   "LIST_CODE_CHAR".Contain_In_Bath11 := "LIST_CODE_CHAR".Contain_In_Bath10;
   "LIST_CODE_CHAR".Contain_In_Bath10 := "LIST_CODE_CHAR".Contain_In_Bath9;
   "LIST_CODE_CHAR".Contain_In_Bath9 := "LIST_CODE_CHAR".Contain_In_Bath8;
   "LIST_CODE_CHAR".Contain_In_Bath8 := "LIST_CODE_CHAR".Contain_In_Bath7;
   "LIST_CODE_CHAR".Contain_In_Bath7 := "LIST_CODE_CHAR".Contain_In_Bath6;
   IF "LIST_CODE_CHAR".Contain_In_Bath6.Barcode_P1 <> '' OR "LIST_CODE_CHAR".Contain_In_Bath6.Barcode_P2 <> '' THEN
       ;
       "LIST_CODE_CHAR".Contain_In_Bath6.Barcode_P1 := '';
       "LIST_CODE_CHAR".Contain_In_Bath6.Barcode_P2 := '';
   END_IF;
   IF "LIST_CODE_CHAR".Contain_In_Bath11.Barcode_P1 <> '' THEN
       ;
       "TCP_PARAMETER".DATA := 'd';
       "SEND_TCP_TRIGGER_1" := TRUE;
   END_IF;


   //Area Robot
   IF "LIST_CODE_CHAR".Contain_In_Bath3.Barcode_P2 = '1' THEN
       ;
       "LIST_CODE_CHAR".Barcode_Queue_Robot := "LIST_CODE_CHAR".Contain_In_Bath3;// Pick to bath 6
       "RUN_TIME_PARAM".REQUEST_PICK_TYPE := 1;
   ELSIF "LIST_CODE_CHAR".Contain_In_Bath3.Barcode_P2 = '2' OR "LIST_CODE_CHAR".Contain_In_Bath3.Barcode_P2 = '3' THEN
       ;
       "LIST_CODE_CHAR".Barcode_Queue_Robot := "LIST_CODE_CHAR".Contain_In_Bath3;// At Bath 4
       "RUN_TIME_PARAM".REQUEST_PICK_TYPE := 3;
   ELSIF "LIST_CODE_CHAR".Contain_In_Bath3.Barcode_P2 = '4' THEN
       ;
       "LIST_CODE_CHAR".Barcode_Queue_Robot := "LIST_CODE_CHAR".Contain_In_Bath3;// Pick To Bath 5
       "RUN_TIME_PARAM".REQUEST_PICK_TYPE := 2;
   ELSE
       "LIST_CODE_CHAR".Barcode_Queue_Robot.Barcode_P1 := '';
       "LIST_CODE_CHAR".Barcode_Queue_Robot.Barcode_P2 := '';
       "RUN_TIME_PARAM".REQUEST_PICK_TYPE := 0;
       ;
   END_IF;

   "LIST_CODE_CHAR".Contain_In_Bath3 := "LIST_CODE_CHAR".Contain_In_Bath2;
   "LIST_CODE_CHAR".Contain_In_Bath2 := "LIST_CODE_CHAR".Contain_In_Bath1;

   // Area 1
   IF "DETECT_VALUE".SCANED_BARCODE <> '' AND "SS Up XL Nâng Input" = TRUE THEN
       ;
       "QUEUE_TO_RUN_BARCODE"(Scaned_Barcode:="DETECT_VALUE".SCANED_BARCODE,OUT_OF_BARCODE=> #Check_Has_Barcode);

   ELSE
       ;
       "LIST_CODE_CHAR".Contain_In_Bath1.Barcode_P1 := '';
       "LIST_CODE_CHAR".Contain_In_Bath1.Barcode_P2 := '';
   END_IF;

   IF #Check_Has_Barcode = TRUE THEN
       ;
       "TCP_PARAMETER".DATA := 'e'; // Khi Không còn barcode trong hàng chờ
       "SEND_TCP_TRIGGER" := TRUE;
   END_IF;
END_FUNCTION

FUNCTION "CONTROL_WATER_PUMP" : Void   // FC2, LAD
{ S7_Optimized_Access := 'TRUE' }
VERSION : 0.1
   VAR_TEMP   // added for the SCL form of the ladder/FBD networks
      _w1 : Bool;
   END_VAR
BEGIN

REGION Network 1: TANK 1
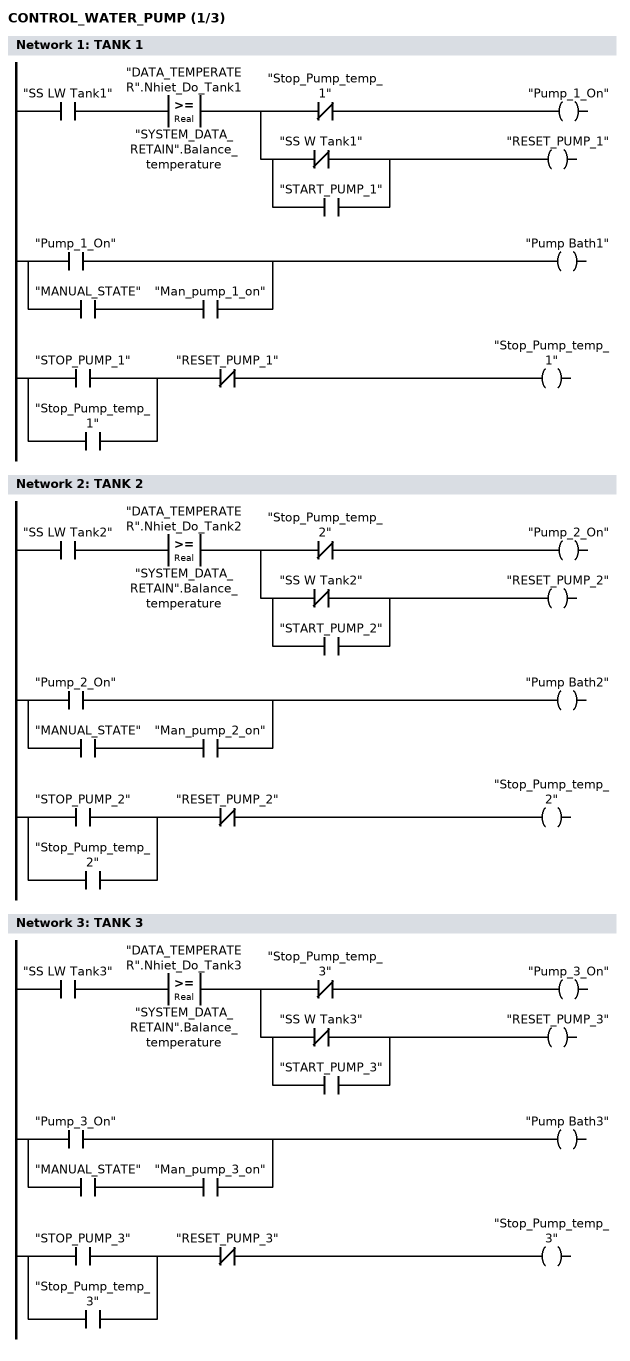
   RUNG wire#powerrail
      Contact( "SS LW Tank1" )
      { S7_Templates := "SrcType := Real" } GE_Contact(in1 := "DATA_TEMPERATER".Nhiet_Do_Tank1, in2 := "SYSTEM_DATA_RETAIN".Balance_temperature)
      wire#w1
      I_Contact( "Stop_Pump_temp_1" )
      Coil( "Pump_1_On" )
   END_RUNG
   RUNG wire#w1
      I_Contact( "SS W Tank1" )
      wire#w2
      Coil( "RESET_PUMP_1" )
   END_RUNG
   RUNG wire#w1
      Contact( "START_PUMP_1" )
   END_RUNG wire#w2
   RUNG wire#powerrail
      Contact( "Pump_1_On" )
      wire#w3
      Coil( "Pump Bath1" )
   END_RUNG
   RUNG wire#powerrail
      Contact( "MANUAL_STATE" )
      Contact( "Man_pump_1_on" )
   END_RUNG wire#w3
   RUNG wire#powerrail
      Contact( "STOP_PUMP_1" )
      wire#w4
      I_Contact( "RESET_PUMP_1" )
      Coil( "Stop_Pump_temp_1" )
   END_RUNG
   RUNG wire#powerrail
      Contact( "Stop_Pump_temp_1" )
   END_RUNG wire#w4
   // the same network as SCL:
   #_w1 := "SS LW Tank1" AND ("DATA_TEMPERATER".Nhiet_Do_Tank1 >= "SYSTEM_DATA_RETAIN".Balance_temperature);
   "Pump_1_On" := #_w1 AND NOT "Stop_Pump_temp_1";
   "RESET_PUMP_1" := #_w1 AND (NOT "SS W Tank1" OR "START_PUMP_1");
   "Pump Bath1" := "Pump_1_On" OR ("MANUAL_STATE" AND "Man_pump_1_on");
   "Stop_Pump_temp_1" := ("STOP_PUMP_1" OR "Stop_Pump_temp_1") AND NOT "RESET_PUMP_1";
END_REGION

REGION Network 2: TANK 2
   RUNG wire#powerrail
      Contact( "SS LW Tank2" )
      { S7_Templates := "SrcType := Real" } GE_Contact(in1 := "DATA_TEMPERATER".Nhiet_Do_Tank2, in2 := "SYSTEM_DATA_RETAIN".Balance_temperature)
      wire#w1
      I_Contact( "Stop_Pump_temp_2" )
      Coil( "Pump_2_On" )
   END_RUNG
   RUNG wire#w1
      I_Contact( "SS W Tank2" )
      wire#w2
      Coil( "RESET_PUMP_2" )
   END_RUNG
   RUNG wire#w1
      Contact( "START_PUMP_2" )
   END_RUNG wire#w2
   RUNG wire#powerrail
      Contact( "Pump_2_On" )
      wire#w3
      Coil( "Pump Bath2" )
   END_RUNG
   RUNG wire#powerrail
      Contact( "MANUAL_STATE" )
      Contact( "Man_pump_2_on" )
   END_RUNG wire#w3
   RUNG wire#powerrail
      Contact( "STOP_PUMP_2" )
      wire#w4
      I_Contact( "RESET_PUMP_2" )
      Coil( "Stop_Pump_temp_2" )
   END_RUNG
   RUNG wire#powerrail
      Contact( "Stop_Pump_temp_2" )
   END_RUNG wire#w4
   // the same network as SCL:
   #_w1 := "SS LW Tank2" AND ("DATA_TEMPERATER".Nhiet_Do_Tank2 >= "SYSTEM_DATA_RETAIN".Balance_temperature);
   "Pump_2_On" := #_w1 AND NOT "Stop_Pump_temp_2";
   "RESET_PUMP_2" := #_w1 AND (NOT "SS W Tank2" OR "START_PUMP_2");
   "Pump Bath2" := "Pump_2_On" OR ("MANUAL_STATE" AND "Man_pump_2_on");
   "Stop_Pump_temp_2" := ("STOP_PUMP_2" OR "Stop_Pump_temp_2") AND NOT "RESET_PUMP_2";
END_REGION

REGION Network 3: TANK 3
   RUNG wire#powerrail
      Contact( "SS LW Tank3" )
      { S7_Templates := "SrcType := Real" } GE_Contact(in1 := "DATA_TEMPERATER".Nhiet_Do_Tank3, in2 := "SYSTEM_DATA_RETAIN".Balance_temperature)
      wire#w1
      I_Contact( "Stop_Pump_temp_3" )
      Coil( "Pump_3_On" )
   END_RUNG
   RUNG wire#w1
      I_Contact( "SS W Tank3" )
      wire#w2
      Coil( "RESET_PUMP_3" )
   END_RUNG
   RUNG wire#w1
      Contact( "START_PUMP_3" )
   END_RUNG wire#w2
   RUNG wire#powerrail
      Contact( "Pump_3_On" )
      wire#w3
      Coil( "Pump Bath3" )
   END_RUNG
   RUNG wire#powerrail
      Contact( "MANUAL_STATE" )
      Contact( "Man_pump_3_on" )
   END_RUNG wire#w3
   RUNG wire#powerrail
      Contact( "STOP_PUMP_3" )
      wire#w4
      I_Contact( "RESET_PUMP_3" )
      Coil( "Stop_Pump_temp_3" )
   END_RUNG
   RUNG wire#powerrail
      Contact( "Stop_Pump_temp_3" )
   END_RUNG wire#w4
   // the same network as SCL:
   #_w1 := "SS LW Tank3" AND ("DATA_TEMPERATER".Nhiet_Do_Tank3 >= "SYSTEM_DATA_RETAIN".Balance_temperature);
   "Pump_3_On" := #_w1 AND NOT "Stop_Pump_temp_3";
   "RESET_PUMP_3" := #_w1 AND (NOT "SS W Tank3" OR "START_PUMP_3");
   "Pump Bath3" := "Pump_3_On" OR ("MANUAL_STATE" AND "Man_pump_3_on");
   "Stop_Pump_temp_3" := ("STOP_PUMP_3" OR "Stop_Pump_temp_3") AND NOT "RESET_PUMP_3";
END_REGION

REGION Network 4: TANK 4
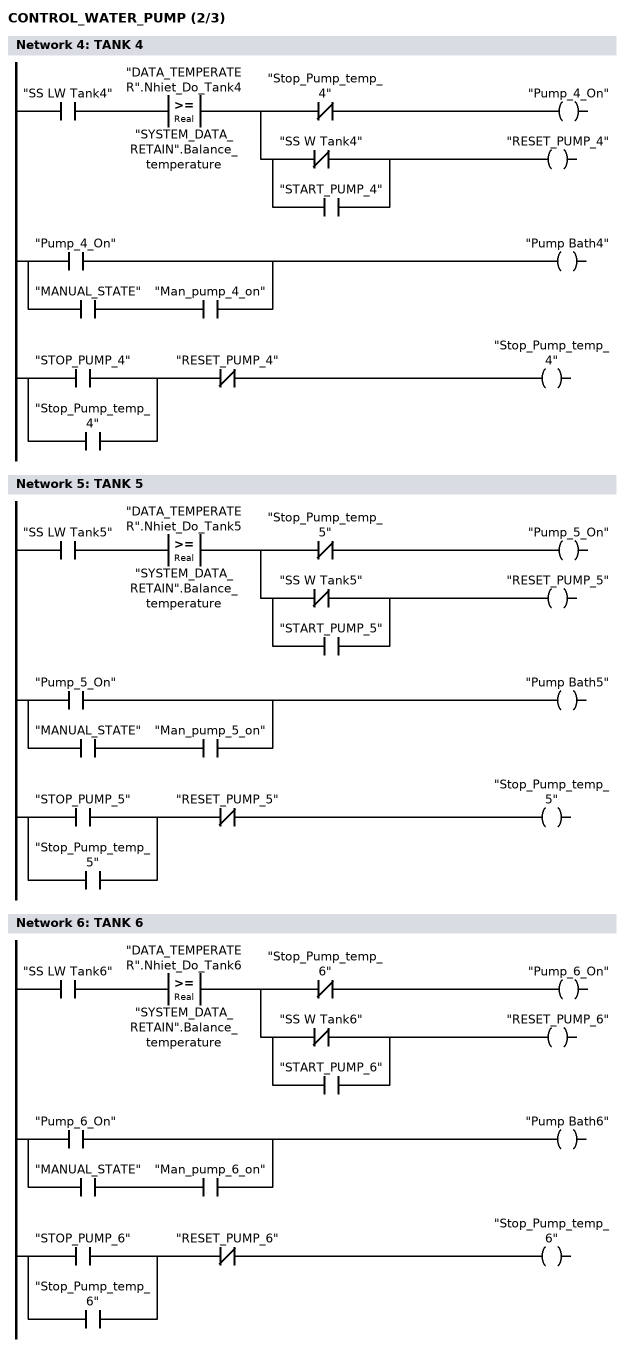
   RUNG wire#powerrail
      Contact( "SS LW Tank4" )
      { S7_Templates := "SrcType := Real" } GE_Contact(in1 := "DATA_TEMPERATER".Nhiet_Do_Tank4, in2 := "SYSTEM_DATA_RETAIN".Balance_temperature)
      wire#w1
      I_Contact( "Stop_Pump_temp_4" )
      Coil( "Pump_4_On" )
   END_RUNG
   RUNG wire#w1
      I_Contact( "SS W Tank4" )
      wire#w2
      Coil( "RESET_PUMP_4" )
   END_RUNG
   RUNG wire#w1
      Contact( "START_PUMP_4" )
   END_RUNG wire#w2
   RUNG wire#powerrail
      Contact( "Pump_4_On" )
      wire#w3
      Coil( "Pump Bath4" )
   END_RUNG
   RUNG wire#powerrail
      Contact( "MANUAL_STATE" )
      Contact( "Man_pump_4_on" )
   END_RUNG wire#w3
   RUNG wire#powerrail
      Contact( "STOP_PUMP_4" )
      wire#w4
      I_Contact( "RESET_PUMP_4" )
      Coil( "Stop_Pump_temp_4" )
   END_RUNG
   RUNG wire#powerrail
      Contact( "Stop_Pump_temp_4" )
   END_RUNG wire#w4
   // the same network as SCL:
   #_w1 := "SS LW Tank4" AND ("DATA_TEMPERATER".Nhiet_Do_Tank4 >= "SYSTEM_DATA_RETAIN".Balance_temperature);
   "Pump_4_On" := #_w1 AND NOT "Stop_Pump_temp_4";
   "RESET_PUMP_4" := #_w1 AND (NOT "SS W Tank4" OR "START_PUMP_4");
   "Pump Bath4" := "Pump_4_On" OR ("MANUAL_STATE" AND "Man_pump_4_on");
   "Stop_Pump_temp_4" := ("STOP_PUMP_4" OR "Stop_Pump_temp_4") AND NOT "RESET_PUMP_4";
END_REGION

REGION Network 5: TANK 5
   RUNG wire#powerrail
      Contact( "SS LW Tank5" )
      { S7_Templates := "SrcType := Real" } GE_Contact(in1 := "DATA_TEMPERATER".Nhiet_Do_Tank5, in2 := "SYSTEM_DATA_RETAIN".Balance_temperature)
      wire#w1
      I_Contact( "Stop_Pump_temp_5" )
      Coil( "Pump_5_On" )
   END_RUNG
   RUNG wire#w1
      I_Contact( "SS W Tank5" )
      wire#w2
      Coil( "RESET_PUMP_5" )
   END_RUNG
   RUNG wire#w1
      Contact( "START_PUMP_5" )
   END_RUNG wire#w2
   RUNG wire#powerrail
      Contact( "Pump_5_On" )
      wire#w3
      Coil( "Pump Bath5" )
   END_RUNG
   RUNG wire#powerrail
      Contact( "MANUAL_STATE" )
      Contact( "Man_pump_5_on" )
   END_RUNG wire#w3
   RUNG wire#powerrail
      Contact( "STOP_PUMP_5" )
      wire#w4
      I_Contact( "RESET_PUMP_5" )
      Coil( "Stop_Pump_temp_5" )
   END_RUNG
   RUNG wire#powerrail
      Contact( "Stop_Pump_temp_5" )
   END_RUNG wire#w4
   // the same network as SCL:
   #_w1 := "SS LW Tank5" AND ("DATA_TEMPERATER".Nhiet_Do_Tank5 >= "SYSTEM_DATA_RETAIN".Balance_temperature);
   "Pump_5_On" := #_w1 AND NOT "Stop_Pump_temp_5";
   "RESET_PUMP_5" := #_w1 AND (NOT "SS W Tank5" OR "START_PUMP_5");
   "Pump Bath5" := "Pump_5_On" OR ("MANUAL_STATE" AND "Man_pump_5_on");
   "Stop_Pump_temp_5" := ("STOP_PUMP_5" OR "Stop_Pump_temp_5") AND NOT "RESET_PUMP_5";
END_REGION

REGION Network 6: TANK 6
   RUNG wire#powerrail
      Contact( "SS LW Tank6" )
      { S7_Templates := "SrcType := Real" } GE_Contact(in1 := "DATA_TEMPERATER".Nhiet_Do_Tank6, in2 := "SYSTEM_DATA_RETAIN".Balance_temperature)
      wire#w1
      I_Contact( "Stop_Pump_temp_6" )
      Coil( "Pump_6_On" )
   END_RUNG
   RUNG wire#w1
      I_Contact( "SS W Tank6" )
      wire#w2
      Coil( "RESET_PUMP_6" )
   END_RUNG
   RUNG wire#w1
      Contact( "START_PUMP_6" )
   END_RUNG wire#w2
   RUNG wire#powerrail
      Contact( "Pump_6_On" )
      wire#w3
      Coil( "Pump Bath6" )
   END_RUNG
   RUNG wire#powerrail
      Contact( "MANUAL_STATE" )
      Contact( "Man_pump_6_on" )
   END_RUNG wire#w3
   RUNG wire#powerrail
      Contact( "STOP_PUMP_6" )
      wire#w4
      I_Contact( "RESET_PUMP_6" )
      Coil( "Stop_Pump_temp_6" )
   END_RUNG
   RUNG wire#powerrail
      Contact( "Stop_Pump_temp_6" )
   END_RUNG wire#w4
   // the same network as SCL:
   #_w1 := "SS LW Tank6" AND ("DATA_TEMPERATER".Nhiet_Do_Tank6 >= "SYSTEM_DATA_RETAIN".Balance_temperature);
   "Pump_6_On" := #_w1 AND NOT "Stop_Pump_temp_6";
   "RESET_PUMP_6" := #_w1 AND (NOT "SS W Tank6" OR "START_PUMP_6");
   "Pump Bath6" := "Pump_6_On" OR ("MANUAL_STATE" AND "Man_pump_6_on");
   "Stop_Pump_temp_6" := ("STOP_PUMP_6" OR "Stop_Pump_temp_6") AND NOT "RESET_PUMP_6";
END_REGION

REGION Network 7: TANK 7
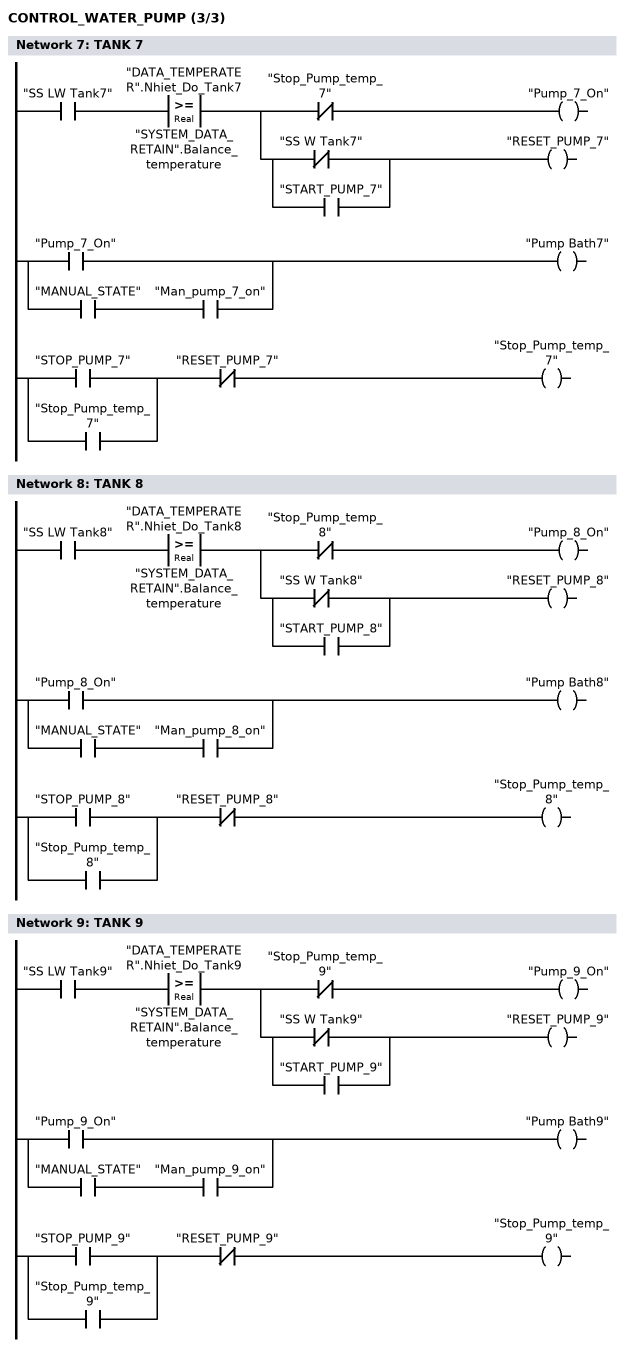
   RUNG wire#powerrail
      Contact( "SS LW Tank7" )
      { S7_Templates := "SrcType := Real" } GE_Contact(in1 := "DATA_TEMPERATER".Nhiet_Do_Tank7, in2 := "SYSTEM_DATA_RETAIN".Balance_temperature)
      wire#w1
      I_Contact( "Stop_Pump_temp_7" )
      Coil( "Pump_7_On" )
   END_RUNG
   RUNG wire#w1
      I_Contact( "SS W Tank7" )
      wire#w2
      Coil( "RESET_PUMP_7" )
   END_RUNG
   RUNG wire#w1
      Contact( "START_PUMP_7" )
   END_RUNG wire#w2
   RUNG wire#powerrail
      Contact( "Pump_7_On" )
      wire#w3
      Coil( "Pump Bath7" )
   END_RUNG
   RUNG wire#powerrail
      Contact( "MANUAL_STATE" )
      Contact( "Man_pump_7_on" )
   END_RUNG wire#w3
   RUNG wire#powerrail
      Contact( "STOP_PUMP_7" )
      wire#w4
      I_Contact( "RESET_PUMP_7" )
      Coil( "Stop_Pump_temp_7" )
   END_RUNG
   RUNG wire#powerrail
      Contact( "Stop_Pump_temp_7" )
   END_RUNG wire#w4
   // the same network as SCL:
   #_w1 := "SS LW Tank7" AND ("DATA_TEMPERATER".Nhiet_Do_Tank7 >= "SYSTEM_DATA_RETAIN".Balance_temperature);
   "Pump_7_On" := #_w1 AND NOT "Stop_Pump_temp_7";
   "RESET_PUMP_7" := #_w1 AND (NOT "SS W Tank7" OR "START_PUMP_7");
   "Pump Bath7" := "Pump_7_On" OR ("MANUAL_STATE" AND "Man_pump_7_on");
   "Stop_Pump_temp_7" := ("STOP_PUMP_7" OR "Stop_Pump_temp_7") AND NOT "RESET_PUMP_7";
END_REGION

REGION Network 8: TANK 8
   RUNG wire#powerrail
      Contact( "SS LW Tank8" )
      { S7_Templates := "SrcType := Real" } GE_Contact(in1 := "DATA_TEMPERATER".Nhiet_Do_Tank8, in2 := "SYSTEM_DATA_RETAIN".Balance_temperature)
      wire#w1
      I_Contact( "Stop_Pump_temp_8" )
      Coil( "Pump_8_On" )
   END_RUNG
   RUNG wire#w1
      I_Contact( "SS W Tank8" )
      wire#w2
      Coil( "RESET_PUMP_8" )
   END_RUNG
   RUNG wire#w1
      Contact( "START_PUMP_8" )
   END_RUNG wire#w2
   RUNG wire#powerrail
      Contact( "Pump_8_On" )
      wire#w3
      Coil( "Pump Bath8" )
   END_RUNG
   RUNG wire#powerrail
      Contact( "MANUAL_STATE" )
      Contact( "Man_pump_8_on" )
   END_RUNG wire#w3
   RUNG wire#powerrail
      Contact( "STOP_PUMP_8" )
      wire#w4
      I_Contact( "RESET_PUMP_8" )
      Coil( "Stop_Pump_temp_8" )
   END_RUNG
   RUNG wire#powerrail
      Contact( "Stop_Pump_temp_8" )
   END_RUNG wire#w4
   // the same network as SCL:
   #_w1 := "SS LW Tank8" AND ("DATA_TEMPERATER".Nhiet_Do_Tank8 >= "SYSTEM_DATA_RETAIN".Balance_temperature);
   "Pump_8_On" := #_w1 AND NOT "Stop_Pump_temp_8";
   "RESET_PUMP_8" := #_w1 AND (NOT "SS W Tank8" OR "START_PUMP_8");
   "Pump Bath8" := "Pump_8_On" OR ("MANUAL_STATE" AND "Man_pump_8_on");
   "Stop_Pump_temp_8" := ("STOP_PUMP_8" OR "Stop_Pump_temp_8") AND NOT "RESET_PUMP_8";
END_REGION

REGION Network 9: TANK 9
   RUNG wire#powerrail
      Contact( "SS LW Tank9" )
      { S7_Templates := "SrcType := Real" } GE_Contact(in1 := "DATA_TEMPERATER".Nhiet_Do_Tank9, in2 := "SYSTEM_DATA_RETAIN".Balance_temperature)
      wire#w1
      I_Contact( "Stop_Pump_temp_9" )
      Coil( "Pump_9_On" )
   END_RUNG
   RUNG wire#w1
      I_Contact( "SS W Tank9" )
      wire#w2
      Coil( "RESET_PUMP_9" )
   END_RUNG
   RUNG wire#w1
      Contact( "START_PUMP_9" )
   END_RUNG wire#w2
   RUNG wire#powerrail
      Contact( "Pump_9_On" )
      wire#w3
      Coil( "Pump Bath9" )
   END_RUNG
   RUNG wire#powerrail
      Contact( "MANUAL_STATE" )
      Contact( "Man_pump_9_on" )
   END_RUNG wire#w3
   RUNG wire#powerrail
      Contact( "STOP_PUMP_9" )
      wire#w4
      I_Contact( "RESET_PUMP_9" )
      Coil( "Stop_Pump_temp_9" )
   END_RUNG
   RUNG wire#powerrail
      Contact( "Stop_Pump_temp_9" )
   END_RUNG wire#w4
   // the same network as SCL:
   #_w1 := "SS LW Tank9" AND ("DATA_TEMPERATER".Nhiet_Do_Tank9 >= "SYSTEM_DATA_RETAIN".Balance_temperature);
   "Pump_9_On" := #_w1 AND NOT "Stop_Pump_temp_9";
   "RESET_PUMP_9" := #_w1 AND (NOT "SS W Tank9" OR "START_PUMP_9");
   "Pump Bath9" := "Pump_9_On" OR ("MANUAL_STATE" AND "Man_pump_9_on");
   "Stop_Pump_temp_9" := ("STOP_PUMP_9" OR "Stop_Pump_temp_9") AND NOT "RESET_PUMP_9";
END_REGION
END_FUNCTION

FUNCTION "Move_BarCode_Data" : Void   // FC3, SCL
{ S7_Optimized_Access := 'TRUE' }
VERSION : 0.1
BEGIN
END_FUNCTION

FUNCTION "INT_TO_BIT_ARRAY" : Void   // FC5, SCL
{ S7_Optimized_Access := 'TRUE' }
VERSION : 0.1
   VAR_INPUT
      IN : Int;
   END_VAR
   VAR_OUTPUT
      OUT : Array[0..15] of Bool;
   END_VAR
   VAR_TEMP
      TEMP : Int;
      TEMPW : Word;
      TEMP_B : Int;
      DEM : Int;
      INS : Int;
   END_VAR
BEGIN
   #TEMP := #IN;
   #TEMP_B := 0;
   #TEMPW := 0;
   #DEM := 0;
   IF #IN = 0 THEN
       FOR #INS := 0 TO 15 DO
           #OUT[#INS] := FALSE;
           ;
       END_FOR;
   ELSE
       WHILE #TEMP <> 0 DO
           #TEMP_B := #TEMP MOD 2;
           #TEMP := #TEMP / 2;
           IF #TEMP_B = 1 THEN
               #OUT[#DEM] := TRUE;
               ;
           ELSIF #TEMP_B = 0 THEN
               #OUT[#DEM] := FALSE;
               ;
           END_IF;
           #DEM := #DEM + 1;
       END_WHILE;
       IF #DEM < 15 THEN
           FOR #DEM := #DEM TO 15 DO
               #OUT[#DEM] := FALSE;
           END_FOR;
       END_IF;
   END_IF;
END_FUNCTION

FUNCTION "QUEUE_TO_RUN_BARCODE" : Void   // FC6, SCL
{ S7_Optimized_Access := 'TRUE' }
VERSION : 0.1
   VAR_INPUT
      Scaned_Barcode : String;
   END_VAR
   VAR_OUTPUT
      OUT_OF_BARCODE : Bool;
   END_VAR
BEGIN
   IF #Scaned_Barcode = "LIST_CODE_CHAR".Barcode_10.Barcode_P1 THEN
       // Truyền barcode vị trí cuối cừng vào ổ chứa barcode ở bể thứ nhất
       "LIST_CODE_CHAR".Contain_In_Bath1 := "LIST_CODE_CHAR".Barcode_10;
       //Reset giá trị Barcode 10 để đẩy mã tiếp theo lên

       //Resort 
       //9->10
       IF "LIST_CODE_CHAR".Barcode_9.Barcode_P1 = '' THEN
           #OUT_OF_BARCODE := TRUE;
       ELSE
           ;
           "LIST_CODE_CHAR".Barcode_10 := "LIST_CODE_CHAR".Barcode_9;
           //8->9
           "LIST_CODE_CHAR".Barcode_9 := "LIST_CODE_CHAR".Barcode_8;
           //7->8
           "LIST_CODE_CHAR".Barcode_8 := "LIST_CODE_CHAR".Barcode_7;
           //6->7
           "LIST_CODE_CHAR".Barcode_7 := "LIST_CODE_CHAR".Barcode_6;
           //5->6
           "LIST_CODE_CHAR".Barcode_6 := "LIST_CODE_CHAR".Barcode_5;
           //4->5
           "LIST_CODE_CHAR".Barcode_5 := "LIST_CODE_CHAR".Barcode_4;
           //3->4
           "LIST_CODE_CHAR".Barcode_4 := "LIST_CODE_CHAR".Barcode_3;
           //2->3
           "LIST_CODE_CHAR".Barcode_3 := "LIST_CODE_CHAR".Barcode_2;
           //1->2
           "LIST_CODE_CHAR".Barcode_2 := "LIST_CODE_CHAR".Barcode_1;
           //''->1
           "LIST_CODE_CHAR".Barcode_1.Barcode_P1 := '';
           "LIST_CODE_CHAR".Barcode_1.Barcode_P2 := '';
           #OUT_OF_BARCODE := FALSE;
       END_IF;

   ELSIF #Scaned_Barcode = "LIST_CODE_CHAR".Barcode_9.Barcode_P1 THEN
       "LIST_CODE_CHAR".Contain_In_Bath1 := "LIST_CODE_CHAR".Barcode_9;
       //Resort
       "LIST_CODE_CHAR".Barcode_9 := "LIST_CODE_CHAR".Barcode_8;
       //7->8
       "LIST_CODE_CHAR".Barcode_8 := "LIST_CODE_CHAR".Barcode_7;
       //6->7
       "LIST_CODE_CHAR".Barcode_7 := "LIST_CODE_CHAR".Barcode_6;
       //5->6
       "LIST_CODE_CHAR".Barcode_6 := "LIST_CODE_CHAR".Barcode_5;
       //4->5
       "LIST_CODE_CHAR".Barcode_5 := "LIST_CODE_CHAR".Barcode_4;
       //3->4
       "LIST_CODE_CHAR".Barcode_4 := "LIST_CODE_CHAR".Barcode_3;
       //2->3
       "LIST_CODE_CHAR".Barcode_3 := "LIST_CODE_CHAR".Barcode_2;
       //1->2
       "LIST_CODE_CHAR".Barcode_2 := "LIST_CODE_CHAR".Barcode_1;
       //''->1
       "LIST_CODE_CHAR".Barcode_1.Barcode_P1 := '';
       "LIST_CODE_CHAR".Barcode_1.Barcode_P2 := '';
       #OUT_OF_BARCODE := FALSE;
   ELSIF #Scaned_Barcode = "LIST_CODE_CHAR".Barcode_8.Barcode_P1 THEN
       "LIST_CODE_CHAR".Contain_In_Bath1 := "LIST_CODE_CHAR".Barcode_8;
       //Resort
       //7->8
       "LIST_CODE_CHAR".Barcode_8 := "LIST_CODE_CHAR".Barcode_7;
       //6->7
       "LIST_CODE_CHAR".Barcode_7 := "LIST_CODE_CHAR".Barcode_6;
       //5->6
       "LIST_CODE_CHAR".Barcode_6 := "LIST_CODE_CHAR".Barcode_5;
       //4->5
       "LIST_CODE_CHAR".Barcode_5 := "LIST_CODE_CHAR".Barcode_4;
       //3->4
       "LIST_CODE_CHAR".Barcode_4 := "LIST_CODE_CHAR".Barcode_3;
       //2->3
       "LIST_CODE_CHAR".Barcode_3 := "LIST_CODE_CHAR".Barcode_2;
       //1->2
       "LIST_CODE_CHAR".Barcode_2 := "LIST_CODE_CHAR".Barcode_1;
       //''->1
       "LIST_CODE_CHAR".Barcode_1.Barcode_P1 := '';
       "LIST_CODE_CHAR".Barcode_1.Barcode_P2 := '';
       #OUT_OF_BARCODE := FALSE;
   ELSIF #Scaned_Barcode = "LIST_CODE_CHAR".Barcode_7.Barcode_P1 THEN
       "LIST_CODE_CHAR".Contain_In_Bath1 := "LIST_CODE_CHAR".Barcode_7;
       //Resort
       //6->7
       "LIST_CODE_CHAR".Barcode_7 := "LIST_CODE_CHAR".Barcode_6;
       //5->6
       "LIST_CODE_CHAR".Barcode_6 := "LIST_CODE_CHAR".Barcode_5;
       //4->5
       "LIST_CODE_CHAR".Barcode_5 := "LIST_CODE_CHAR".Barcode_4;
       //3->4
       "LIST_CODE_CHAR".Barcode_4 := "LIST_CODE_CHAR".Barcode_3;
       //2->3
       "LIST_CODE_CHAR".Barcode_3 := "LIST_CODE_CHAR".Barcode_2;
       //1->2
       "LIST_CODE_CHAR".Barcode_2 := "LIST_CODE_CHAR".Barcode_1;
       //''->1
       "LIST_CODE_CHAR".Barcode_1.Barcode_P1 := '';
       "LIST_CODE_CHAR".Barcode_1.Barcode_P2 := '';
       #OUT_OF_BARCODE := FALSE;
   ELSIF #Scaned_Barcode = "LIST_CODE_CHAR".Barcode_6.Barcode_P1 THEN
       "LIST_CODE_CHAR".Contain_In_Bath1 := "LIST_CODE_CHAR".Barcode_6;
       //Resort
       //5->6
       "LIST_CODE_CHAR".Barcode_6 := "LIST_CODE_CHAR".Barcode_5;
       //4->5
       "LIST_CODE_CHAR".Barcode_5 := "LIST_CODE_CHAR".Barcode_4;
       //3->4
       "LIST_CODE_CHAR".Barcode_4 := "LIST_CODE_CHAR".Barcode_3;
       //2->3
       "LIST_CODE_CHAR".Barcode_3 := "LIST_CODE_CHAR".Barcode_2;
       //1->2
       "LIST_CODE_CHAR".Barcode_2 := "LIST_CODE_CHAR".Barcode_1;
       //''->1
       "LIST_CODE_CHAR".Barcode_1.Barcode_P1 := '';
       "LIST_CODE_CHAR".Barcode_1.Barcode_P2 := '';
       #OUT_OF_BARCODE := FALSE;
   ELSIF #Scaned_Barcode = "LIST_CODE_CHAR".Barcode_5.Barcode_P1 THEN
       "LIST_CODE_CHAR".Contain_In_Bath1 := "LIST_CODE_CHAR".Barcode_5;
       //Resort
       //4->5
       "LIST_CODE_CHAR".Barcode_5 := "LIST_CODE_CHAR".Barcode_4;
       //3->4
       "LIST_CODE_CHAR".Barcode_4 := "LIST_CODE_CHAR".Barcode_3;
       //2->3
       "LIST_CODE_CHAR".Barcode_3 := "LIST_CODE_CHAR".Barcode_2;
       //1->2
       "LIST_CODE_CHAR".Barcode_2 := "LIST_CODE_CHAR".Barcode_1;
       //''->1
       "LIST_CODE_CHAR".Barcode_1.Barcode_P1 := '';
       "LIST_CODE_CHAR".Barcode_1.Barcode_P2 := '';
       #OUT_OF_BARCODE := FALSE;
   ELSIF #Scaned_Barcode = "LIST_CODE_CHAR".Barcode_4.Barcode_P1 THEN
       "LIST_CODE_CHAR".Contain_In_Bath1 := "LIST_CODE_CHAR".Barcode_4;
       //Resort
       //3->4
       "LIST_CODE_CHAR".Barcode_4 := "LIST_CODE_CHAR".Barcode_3;
       //2->3
       "LIST_CODE_CHAR".Barcode_3 := "LIST_CODE_CHAR".Barcode_2;
       //1->2
       "LIST_CODE_CHAR".Barcode_2 := "LIST_CODE_CHAR".Barcode_1;
       //''->1
       "LIST_CODE_CHAR".Barcode_1.Barcode_P1 := '';
       "LIST_CODE_CHAR".Barcode_1.Barcode_P2 := '';
       #OUT_OF_BARCODE := FALSE;
   ELSIF #Scaned_Barcode = "LIST_CODE_CHAR".Barcode_3.Barcode_P1 THEN
       "LIST_CODE_CHAR".Contain_In_Bath1 := "LIST_CODE_CHAR".Barcode_3;
       //Resort
       //2->3
       "LIST_CODE_CHAR".Barcode_3 := "LIST_CODE_CHAR".Barcode_2;
       //1->2
       "LIST_CODE_CHAR".Barcode_2 := "LIST_CODE_CHAR".Barcode_1;
       //''->1
       "LIST_CODE_CHAR".Barcode_1.Barcode_P1 := '';
       "LIST_CODE_CHAR".Barcode_1.Barcode_P2 := '';
       #OUT_OF_BARCODE := FALSE;
   ELSIF #Scaned_Barcode = "LIST_CODE_CHAR".Barcode_2.Barcode_P1 THEN
       "LIST_CODE_CHAR".Contain_In_Bath1 := "LIST_CODE_CHAR".Barcode_2;
       //Resort
       //1->2
       "LIST_CODE_CHAR".Barcode_2 := "LIST_CODE_CHAR".Barcode_1;
       //''->1
       "LIST_CODE_CHAR".Barcode_1.Barcode_P1 := '';
       "LIST_CODE_CHAR".Barcode_1.Barcode_P2 := '';
       #OUT_OF_BARCODE := FALSE;
   ELSIF #Scaned_Barcode = "LIST_CODE_CHAR".Barcode_1.Barcode_P1 THEN
       "LIST_CODE_CHAR".Contain_In_Bath1 := "LIST_CODE_CHAR".Barcode_1;
       //Resort
       //''->1
       "LIST_CODE_CHAR".Barcode_1.Barcode_P1 := '';
       "LIST_CODE_CHAR".Barcode_1.Barcode_P2 := '';
       #OUT_OF_BARCODE := FALSE;
   END_IF;

   "DETECT_VALUE".INPUT_SCANED_BARCODE := '';
END_FUNCTION

FUNCTION "CheckFirst_Initial_Process" : Void   // FC7, SCL
{ S7_Optimized_Access := 'TRUE' }
VERSION : 0.1
   VAR_OUTPUT
      FIRST_RACK : Bool;
   END_VAR
   VAR_TEMP
      _counter_ : Int;
      isExistRack1 : Bool;
      isExistRack2 : Bool;
      isExistRack3 : Bool;
      isExistRack4 : Bool;
      isExistRack5 : Bool;
      isExistRack6 : Bool;
      isExistRack7 : Bool;
      isExistRack8 : Bool;
      isExistRack9 : Bool;
      isExistRack10 : Bool;
   END_VAR
BEGIN
   #isExistRack1 := TRUE;
   #isExistRack2 := TRUE;
   #isExistRack3 := TRUE;
   #isExistRack4 := TRUE;
   #isExistRack5 := TRUE;
   #isExistRack6 := TRUE;
   #isExistRack7 := TRUE;
   #isExistRack8 := TRUE;
   #isExistRack9 := TRUE;
   #isExistRack10 := TRUE;
   IF "LIST_CODE_CHAR".Contain_In_Bath1.Barcode_P1='' THEN
       // Statement section IF
       #isExistRack1 := FALSE
       ;
   END_IF;
   IF "LIST_CODE_CHAR".Contain_In_Bath2.Barcode_P1 = '' THEN
       // Statement section IF
       #isExistRack2 := FALSE
       ;
   END_IF;
   IF "LIST_CODE_CHAR".Contain_In_Bath3.Barcode_P1 = '' THEN
       // Statement section IF
       #isExistRack3 := FALSE
       ;
   END_IF;
   IF "LIST_CODE_CHAR".Contain_In_Bath4.Barcode_P1 = '' THEN
       // Statement section IF
       #isExistRack4 := FALSE
       ;
   END_IF;
   IF "LIST_CODE_CHAR".Contain_In_Bath5.Barcode_P1 = '' THEN
       // Statement section IF
       #isExistRack5 := FALSE
       ;
   END_IF;
   IF "LIST_CODE_CHAR".Contain_In_Bath6.Barcode_P1 = '' THEN
       // Statement section IF
       #isExistRack6 := FALSE
       ;
   END_IF;
   IF "LIST_CODE_CHAR".Contain_In_Bath7.Barcode_P1 = '' THEN
       // Statement section IF
       #isExistRack7 := FALSE
       ;
   END_IF;
   IF "LIST_CODE_CHAR".Contain_In_Bath8.Barcode_P1 = '' THEN
       // Statement section IF
       #isExistRack8 := FALSE
       ;
   END_IF;
   IF "LIST_CODE_CHAR".Contain_In_Bath9.Barcode_P1 = '' THEN
       // Statement section IF
       #isExistRack9 := FALSE
       ;
   END_IF;
   IF "LIST_CODE_CHAR".Contain_In_Bath10.Barcode_P1 = '' THEN
       // Statement section IF
       #isExistRack10 := FALSE
       ;
   END_IF;

   IF #isExistRack1=FALSE
       & #isExistRack2=FALSE
       & #isExistRack3=FALSE
       & #isExistRack4=FALSE
       & #isExistRack5=FALSE
       & #isExistRack6=FALSE
       & #isExistRack7=FALSE
       & #isExistRack8=FALSE
       & #isExistRack9=FALSE
       & #isExistRack10=FALSE THEN
       #FIRST_RACK := TRUE;
       ;
   ELSE
       #FIRST_RACK:=FALSE
       ;
   END_IF;
END_FUNCTION

ORGANIZATION_BLOCK "Main"   // OB1, LAD, ProgramCycle
TITLE = "Main Program Sweep (Cycle)"
{ S7_Optimized_Access := 'TRUE' }
VERSION : 0.1
   VAR_INPUT
      Initial_Call : Bool;   // Initial call of this OB
      Remanence : Bool;   // =True, if remanent data are available
   END_VAR
   VAR_TEMP   // added for the SCL form of the ladder/FBD networks
      _w1 : Bool;
      _w2 : Bool;
      _w3 : Bool;
      _w4 : Bool;
      _w5 : Bool;
      _w6 : Bool;
      _w7 : Bool;
      _w8 : Bool;
      _w9 : Bool;
      _w10 : Bool;
      _w11 : Bool;
      _w12 : Bool;
      _w13 : Bool;
      _w14 : Bool;
      _w15 : Bool;
      _w16 : Bool;
      _w17 : Bool;
      _w18 : Bool;
      _w19 : Bool;
      _w20 : Bool;
      _w21 : Bool;
      _w22 : Bool;
      _w23 : Bool;
      _w24 : Bool;
      _w25 : Bool;
      _w26 : Bool;
      _w27 : Bool;
      _w28 : Bool;
      _w29 : Bool;
   END_VAR
BEGIN

REGION Network 1: STRT - STOP - RESET Control
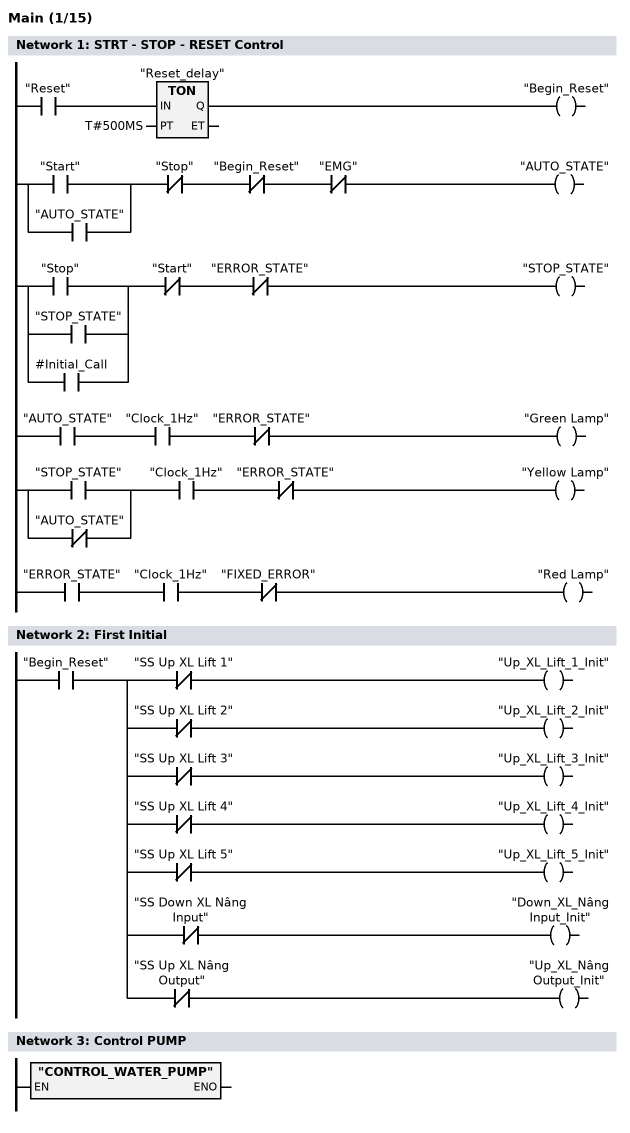
   "Reset_delay".TON(IN := "Reset", PT := T#500MS);
   "Begin_Reset" := "Reset_delay".Q;
   "AUTO_STATE" := ("Start" OR "AUTO_STATE") AND NOT "Stop" AND NOT "Begin_Reset" AND NOT "EMG";
   "STOP_STATE" := ("Stop" OR "STOP_STATE" OR #Initial_Call) AND NOT "Start" AND NOT "ERROR_STATE";
   "Green Lamp" := "AUTO_STATE" AND "Clock_1Hz" AND NOT "ERROR_STATE";
   "Yellow Lamp" := ("STOP_STATE" OR NOT "AUTO_STATE") AND "Clock_1Hz" AND NOT "ERROR_STATE";
   "Red Lamp" := "ERROR_STATE" AND "Clock_1Hz" AND NOT "FIXED_ERROR";
END_REGION

REGION Network 2: First Initial
   RUNG wire#powerrail
      Contact( "Begin_Reset" )
      wire#w1
      I_Contact( "SS Up XL Lift 1" )
      Coil( "Up_XL_Lift_1_Init" )
   END_RUNG
   RUNG wire#w1
      I_Contact( "SS Up XL Lift 2" )
      Coil( "Up_XL_Lift_2_Init" )
   END_RUNG
   RUNG wire#w1
      I_Contact( "SS Up XL Lift 3" )
      Coil( "Up_XL_Lift_3_Init" )
   END_RUNG
   RUNG wire#w1
      I_Contact( "SS Up XL Lift 4" )
      Coil( "Up_XL_Lift_4_Init" )
   END_RUNG
   RUNG wire#w1
      I_Contact( "SS Up XL Lift 5" )
      Coil( "Up_XL_Lift_5_Init" )
   END_RUNG
   RUNG wire#w1
      I_Contact( "SS Down XL Nâng Input" )
      Coil( "Down_XL_Nâng Input_Init" )
   END_RUNG
   RUNG wire#w1
      I_Contact( "SS Up XL Nâng Output" )
      Coil( "Up_XL_Nâng Output_Init" )
   END_RUNG
   // the same network as SCL:
   "Up_XL_Lift_1_Init" := "Begin_Reset" AND NOT "SS Up XL Lift 1";
   "Up_XL_Lift_2_Init" := "Begin_Reset" AND NOT "SS Up XL Lift 2";
   "Up_XL_Lift_3_Init" := "Begin_Reset" AND NOT "SS Up XL Lift 3";
   "Up_XL_Lift_4_Init" := "Begin_Reset" AND NOT "SS Up XL Lift 4";
   "Up_XL_Lift_5_Init" := "Begin_Reset" AND NOT "SS Up XL Lift 5";
   "Down_XL_Nâng Input_Init" := "Begin_Reset" AND NOT "SS Down XL Nâng Input";
   "Up_XL_Nâng Output_Init" := "Begin_Reset" AND NOT "SS Up XL Nâng Output";
END_REGION

REGION Network 3: Control PUMP
   RUNG wire#powerrail
      "CONTROL_WATER_PUMP"()
   END_RUNG
   // the same network as SCL:
   "CONTROL_WATER_PUMP"();
END_REGION

REGION Network 4: Trigger Jog BW Tranfer 1 2
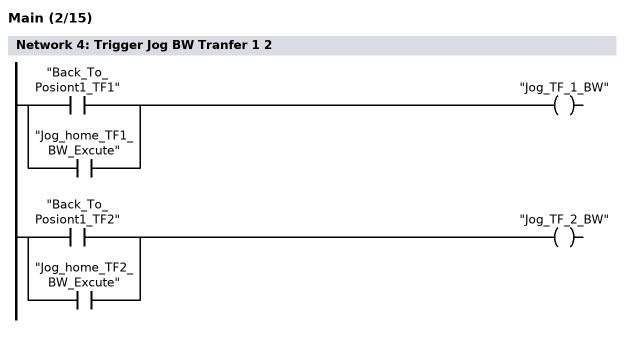
   RUNG wire#powerrail
      Contact( "Back_To_Posiont1_TF1" )
      wire#w1
      Coil( "Jog_TF_1_BW" )
   END_RUNG
   RUNG wire#powerrail
      Contact( "Jog_home_TF1_BW_Excute" )
   END_RUNG wire#w1
   RUNG wire#powerrail
      Contact( "Back_To_Posiont1_TF2" )
      wire#w2
      Coil( "Jog_TF_2_BW" )
   END_RUNG
   RUNG wire#powerrail
      Contact( "Jog_home_TF2_BW_Excute" )
   END_RUNG wire#w2
   // the same network as SCL:
   "Jog_TF_1_BW" := "Back_To_Posiont1_TF1" OR "Jog_home_TF1_BW_Excute";
   "Jog_TF_2_BW" := "Back_To_Posiont1_TF2" OR "Jog_home_TF2_BW_Excute";
END_REGION

REGION Network 5: Initail Tranfer 1 Group
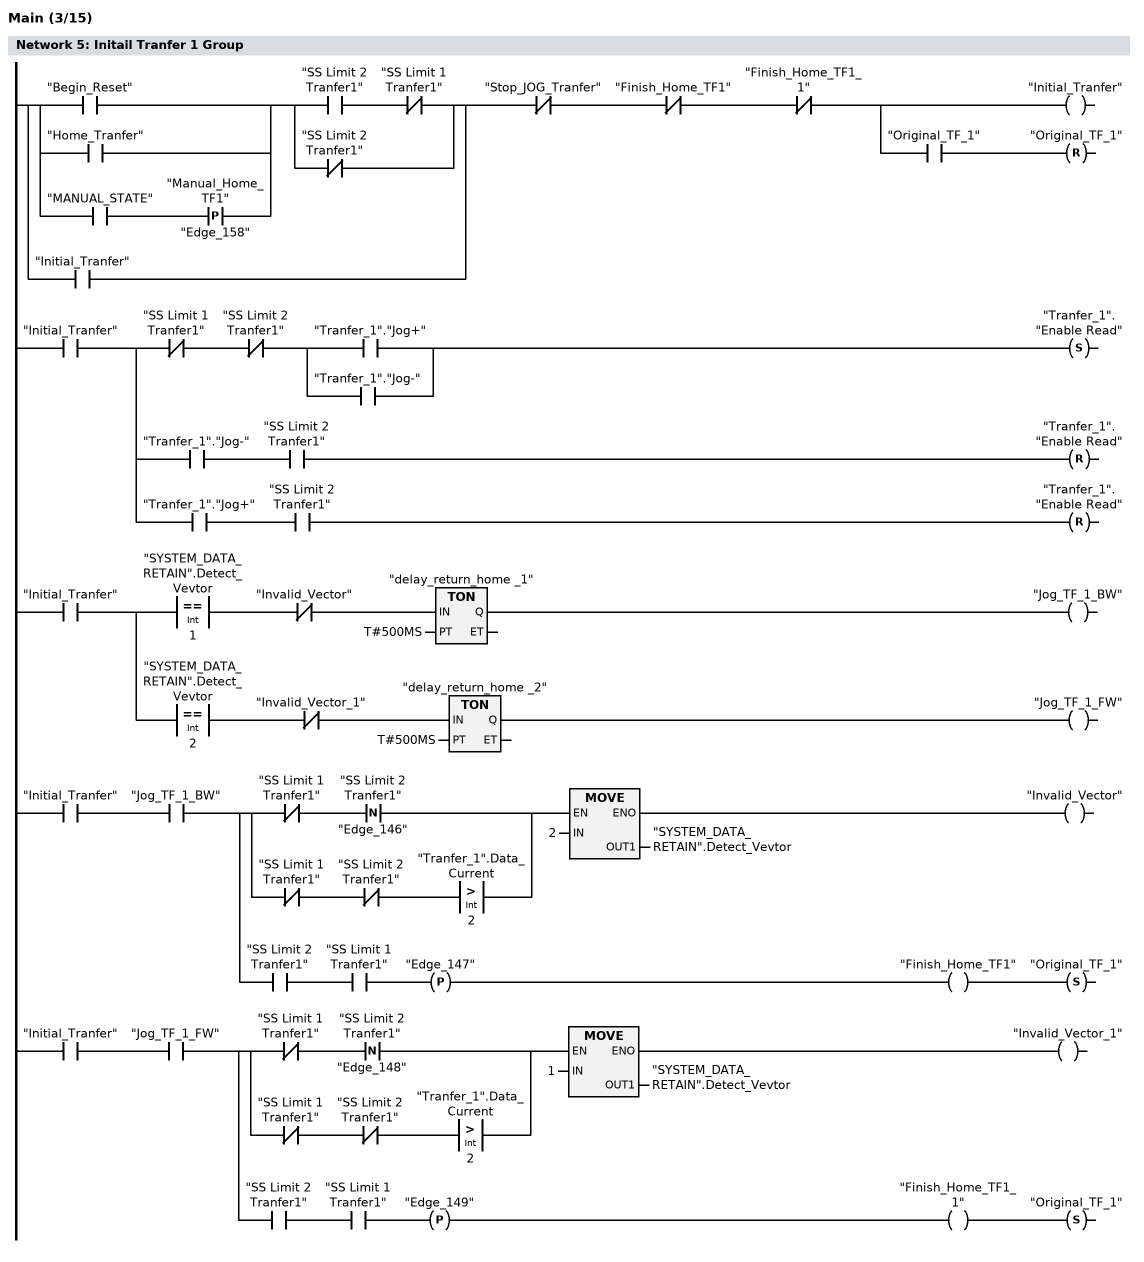
   // ENO of a box is taken as its EN; it also drops when the box reports an error
   #_w1 := "MANUAL_STATE" AND "Manual_Home_TF1" AND NOT "Edge_158";   // rising edge of "Manual_Home_TF1"
   "Edge_158" := "Manual_Home_TF1";
   "Initial_Tranfer" := ((("Begin_Reset" OR "Home_Tranfer" OR #_w1) AND (("SS Limit 2 Tranfer1" AND NOT "SS Limit 1 Tranfer1") OR NOT "SS Limit 2 Tranfer1")) OR "Initial_Tranfer") AND NOT "Stop_JOG_Tranfer" AND NOT "Finish_Home_TF1" AND NOT "Finish_Home_TF1_1";
   IF "Initial_Tranfer" AND "Original_TF_1" THEN "Original_TF_1" := FALSE; END_IF;
   IF "Initial_Tranfer" AND NOT "SS Limit 1 Tranfer1" AND NOT "SS Limit 2 Tranfer1" AND ("Tranfer_1"."Jog+" OR "Tranfer_1"."Jog-") THEN
       "Tranfer_1"."Enable Read" := TRUE;
   END_IF;
   IF "Initial_Tranfer" AND "Tranfer_1"."Jog-" AND "SS Limit 2 Tranfer1" THEN
       "Tranfer_1"."Enable Read" := FALSE;
   END_IF;
   IF "Initial_Tranfer" AND "Tranfer_1"."Jog+" AND "SS Limit 2 Tranfer1" THEN
       "Tranfer_1"."Enable Read" := FALSE;
   END_IF;
   "delay_return_home _1".TON(IN := "Initial_Tranfer" AND ("SYSTEM_DATA_RETAIN".Detect_Vevtor = 1) AND NOT "Invalid_Vector",
                           PT := T#500MS);
   "Jog_TF_1_BW" := "delay_return_home _1".Q;
   "delay_return_home _2".TON(IN := "Initial_Tranfer" AND ("SYSTEM_DATA_RETAIN".Detect_Vevtor = 2) AND NOT "Invalid_Vector_1",
                           PT := T#500MS);
   "Jog_TF_1_FW" := "delay_return_home _2".Q;
   #_w2 := "Initial_Tranfer" AND "Jog_TF_1_BW";
   #_w3 := #_w2 AND NOT "SS Limit 1 Tranfer1" AND NOT "SS Limit 2 Tranfer1" AND "Edge_146";   // falling edge of "SS Limit 2 Tranfer1"
   "Edge_146" := "SS Limit 2 Tranfer1";
   #_w4 := #_w3 OR (#_w2 AND NOT "SS Limit 1 Tranfer1" AND NOT "SS Limit 2 Tranfer1" AND ("Tranfer_1".Data_Current > 2));
   IF #_w4 THEN "SYSTEM_DATA_RETAIN".Detect_Vevtor := 2; END_IF;
   "Invalid_Vector" := #_w4;
   #_w5 := #_w2 AND "SS Limit 2 Tranfer1" AND "SS Limit 1 Tranfer1";
   #_w6 := #_w5 AND NOT "Edge_147";   // rising edge
   "Edge_147" := #_w5;
   "Finish_Home_TF1" := #_w6;
   IF #_w6 THEN "Original_TF_1" := TRUE; END_IF;
   #_w7 := "Initial_Tranfer" AND "Jog_TF_1_FW";
   #_w8 := #_w7 AND NOT "SS Limit 1 Tranfer1" AND NOT "SS Limit 2 Tranfer1" AND "Edge_148";   // falling edge of "SS Limit 2 Tranfer1"
   "Edge_148" := "SS Limit 2 Tranfer1";
   #_w9 := #_w8 OR (#_w7 AND NOT "SS Limit 1 Tranfer1" AND NOT "SS Limit 2 Tranfer1" AND ("Tranfer_1".Data_Current > 2));
   IF #_w9 THEN "SYSTEM_DATA_RETAIN".Detect_Vevtor := 1; END_IF;
   "Invalid_Vector_1" := #_w9;
   #_w10 := #_w7 AND "SS Limit 2 Tranfer1" AND "SS Limit 1 Tranfer1";
   #_w11 := #_w10 AND NOT "Edge_149";   // rising edge
   "Edge_149" := #_w10;
   "Finish_Home_TF1_1" := #_w11;
   IF #_w11 THEN "Original_TF_1" := TRUE; END_IF;
END_REGION

REGION Network 6: Initail Tranfer 2 Group
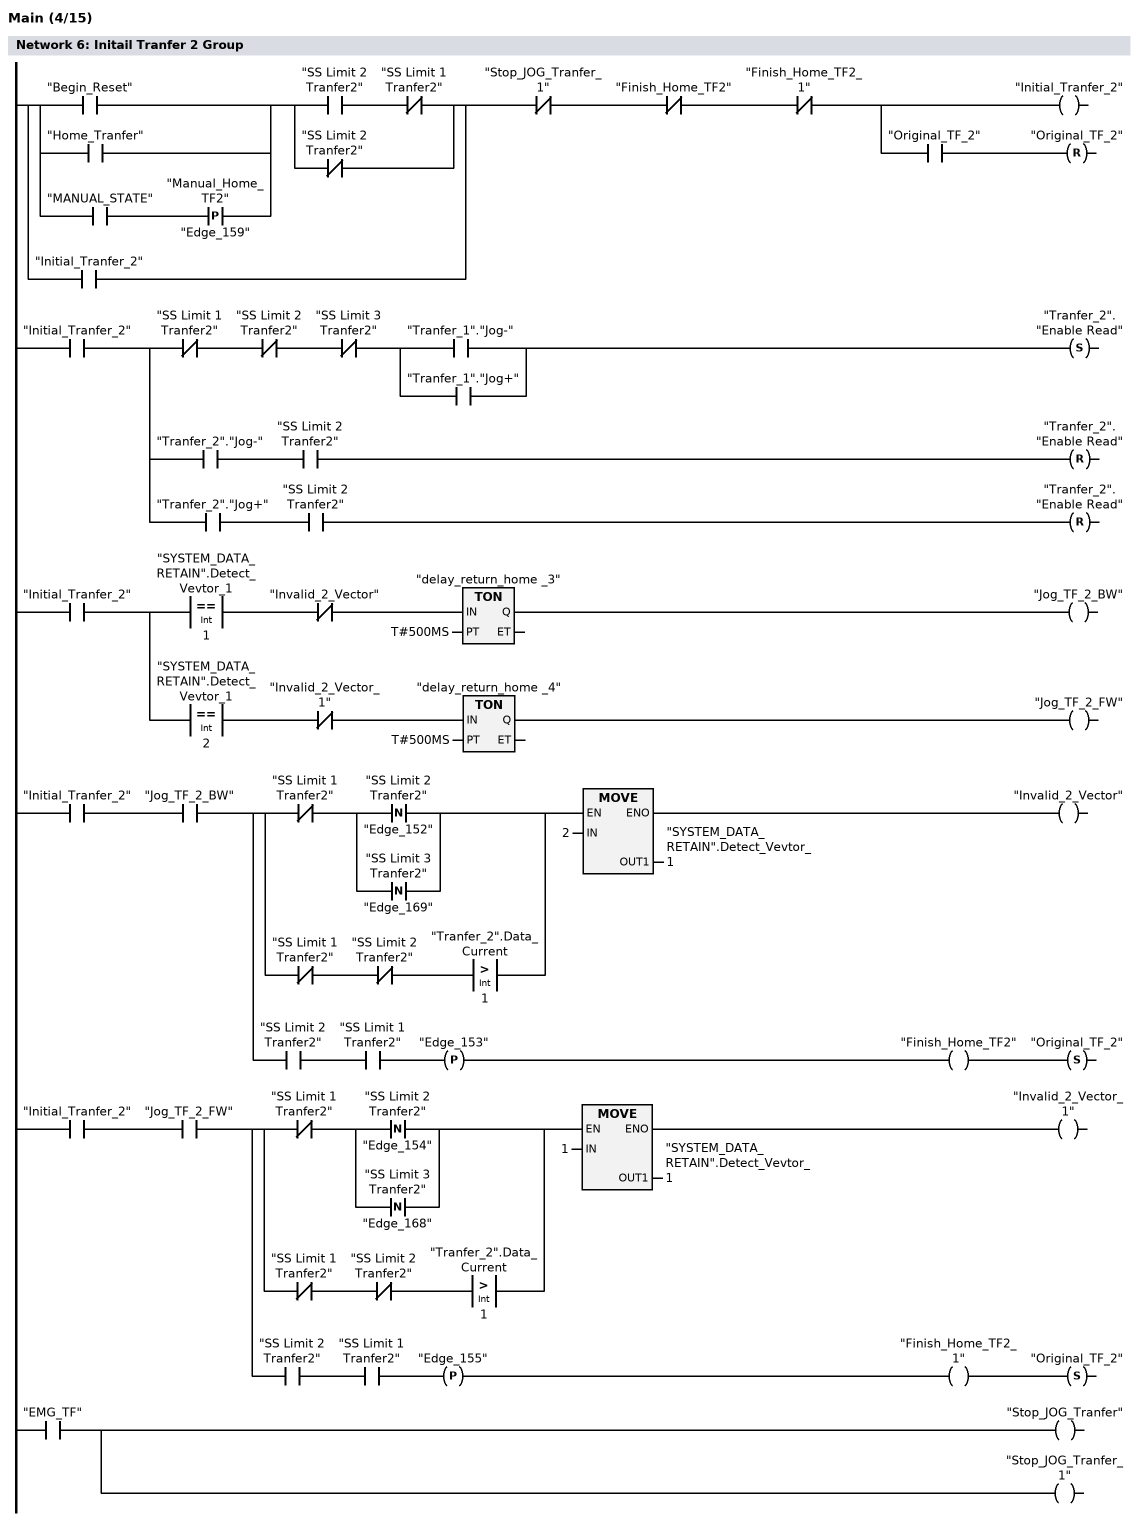
   // ENO of a box is taken as its EN; it also drops when the box reports an error
   #_w1 := "MANUAL_STATE" AND "Manual_Home_TF2" AND NOT "Edge_159";   // rising edge of "Manual_Home_TF2"
   "Edge_159" := "Manual_Home_TF2";
   "Initial_Tranfer_2" := ((("Begin_Reset" OR "Home_Tranfer" OR #_w1) AND (("SS Limit 2 Tranfer2" AND NOT "SS Limit 1 Tranfer2") OR NOT "SS Limit 2 Tranfer2")) OR "Initial_Tranfer_2") AND NOT "Stop_JOG_Tranfer_1" AND NOT "Finish_Home_TF2" AND NOT "Finish_Home_TF2_1";
   IF "Initial_Tranfer_2" AND "Original_TF_2" THEN "Original_TF_2" := FALSE; END_IF;
   IF "Initial_Tranfer_2" AND NOT "SS Limit 1 Tranfer2" AND NOT "SS Limit 2 Tranfer2" AND NOT "SS Limit 3 Tranfer2" AND ("Tranfer_1"."Jog-" OR "Tranfer_1"."Jog+") THEN
       "Tranfer_2"."Enable Read" := TRUE;
   END_IF;
   IF "Initial_Tranfer_2" AND "Tranfer_2"."Jog-" AND "SS Limit 2 Tranfer2" THEN
       "Tranfer_2"."Enable Read" := FALSE;
   END_IF;
   IF "Initial_Tranfer_2" AND "Tranfer_2"."Jog+" AND "SS Limit 2 Tranfer2" THEN
       "Tranfer_2"."Enable Read" := FALSE;
   END_IF;
   "delay_return_home _3".TON(IN := "Initial_Tranfer_2" AND ("SYSTEM_DATA_RETAIN".Detect_Vevtor_1 = 1) AND NOT "Invalid_2_Vector",
                           PT := T#500MS);
   "Jog_TF_2_BW" := "delay_return_home _3".Q;
   "delay_return_home _4".TON(IN := "Initial_Tranfer_2" AND ("SYSTEM_DATA_RETAIN".Detect_Vevtor_1 = 2) AND NOT "Invalid_2_Vector_1",
                           PT := T#500MS);
   "Jog_TF_2_FW" := "delay_return_home _4".Q;
   #_w2 := "Initial_Tranfer_2" AND "Jog_TF_2_BW";
   #_w3 := #_w2 AND NOT "SS Limit 1 Tranfer2" AND NOT "SS Limit 2 Tranfer2" AND "Edge_152";   // falling edge of "SS Limit 2 Tranfer2"
   "Edge_152" := "SS Limit 2 Tranfer2";
   #_w4 := #_w2 AND NOT "SS Limit 1 Tranfer2" AND NOT "SS Limit 3 Tranfer2" AND "Edge_169";   // falling edge of "SS Limit 3 Tranfer2"
   "Edge_169" := "SS Limit 3 Tranfer2";
   #_w5 := #_w3 OR #_w4 OR (#_w2 AND NOT "SS Limit 1 Tranfer2" AND NOT "SS Limit 2 Tranfer2" AND ("Tranfer_2".Data_Current > 1));
   IF #_w5 THEN "SYSTEM_DATA_RETAIN".Detect_Vevtor_1 := 2; END_IF;
   "Invalid_2_Vector" := #_w5;
   #_w6 := #_w2 AND "SS Limit 2 Tranfer2" AND "SS Limit 1 Tranfer2";
   #_w7 := #_w6 AND NOT "Edge_153";   // rising edge
   "Edge_153" := #_w6;
   "Finish_Home_TF2" := #_w7;
   IF #_w7 THEN "Original_TF_2" := TRUE; END_IF;
   #_w8 := "Initial_Tranfer_2" AND "Jog_TF_2_FW";
   #_w9 := #_w8 AND NOT "SS Limit 1 Tranfer2" AND NOT "SS Limit 2 Tranfer2" AND "Edge_154";   // falling edge of "SS Limit 2 Tranfer2"
   "Edge_154" := "SS Limit 2 Tranfer2";
   #_w10 := #_w8 AND NOT "SS Limit 1 Tranfer2" AND NOT "SS Limit 3 Tranfer2" AND "Edge_168";   // falling edge of "SS Limit 3 Tranfer2"
   "Edge_168" := "SS Limit 3 Tranfer2";
   #_w11 := #_w9 OR #_w10 OR (#_w8 AND NOT "SS Limit 1 Tranfer2" AND NOT "SS Limit 2 Tranfer2" AND ("Tranfer_2".Data_Current > 1));
   IF #_w11 THEN "SYSTEM_DATA_RETAIN".Detect_Vevtor_1 := 1; END_IF;
   "Invalid_2_Vector_1" := #_w11;
   #_w12 := #_w8 AND "SS Limit 2 Tranfer2" AND "SS Limit 1 Tranfer2";
   #_w13 := #_w12 AND NOT "Edge_155";   // rising edge
   "Edge_155" := #_w12;
   "Finish_Home_TF2_1" := #_w13;
   IF #_w13 THEN "Original_TF_2" := TRUE; END_IF;
   "Stop_JOG_Tranfer" := "EMG_TF";
   "Stop_JOG_Tranfer_1" := "EMG_TF";
END_REGION

REGION Network 7: Detect Position Tranfer
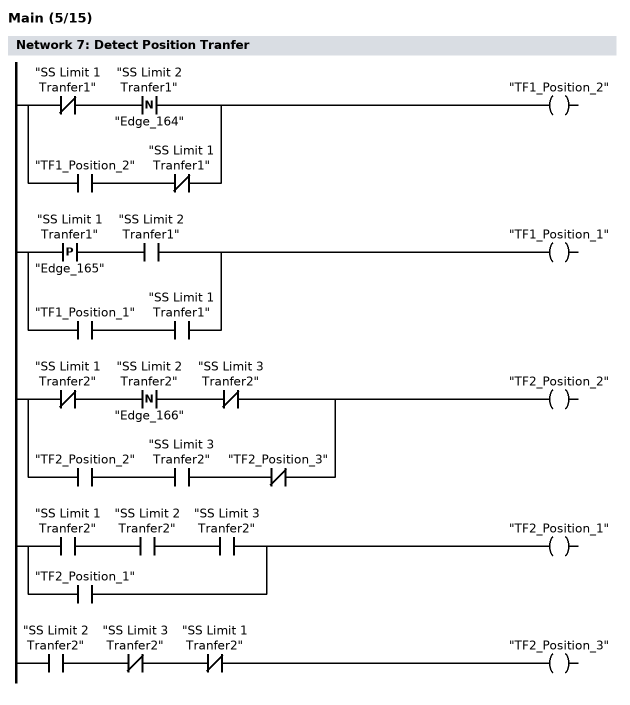
   RUNG wire#powerrail
      I_Contact( "SS Limit 1 Tranfer1" )
      N_Contact(operand := "SS Limit 2 Tranfer1", bit := "Edge_164")
      wire#w1
      Coil( "TF1_Position_2" )
   END_RUNG
   RUNG wire#powerrail
      Contact( "TF1_Position_2" )
      I_Contact( "SS Limit 1 Tranfer1" )
   END_RUNG wire#w1
   RUNG wire#powerrail
      P_Contact(operand := "SS Limit 1 Tranfer1", bit := "Edge_165")
      Contact( "SS Limit 2 Tranfer1" )
      wire#w2
      Coil( "TF1_Position_1" )
   END_RUNG
   RUNG wire#powerrail
      Contact( "TF1_Position_1" )
      Contact( "SS Limit 1 Tranfer1" )
   END_RUNG wire#w2
   RUNG wire#powerrail
      I_Contact( "SS Limit 1 Tranfer2" )
      N_Contact(operand := "SS Limit 2 Tranfer2", bit := "Edge_166")
      I_Contact( "SS Limit 3 Tranfer2" )
      wire#w3
      Coil( "TF2_Position_2" )
   END_RUNG
   RUNG wire#powerrail
      Contact( "TF2_Position_2" )
      Contact( "SS Limit 3 Tranfer2" )
      I_Contact( "TF2_Position_3" )
   END_RUNG wire#w3
   RUNG wire#powerrail
      Contact( "SS Limit 1 Tranfer2" )
      Contact( "SS Limit 2 Tranfer2" )
      Contact( "SS Limit 3 Tranfer2" )
      wire#w4
      Coil( "TF2_Position_1" )
   END_RUNG
   RUNG wire#powerrail
      Contact( "TF2_Position_1" )
   END_RUNG wire#w4
   RUNG wire#powerrail
      Contact( "SS Limit 2 Tranfer2" )
      I_Contact( "SS Limit 3 Tranfer2" )
      I_Contact( "SS Limit 1 Tranfer2" )
      Coil( "TF2_Position_3" )
   END_RUNG
   // the same network as SCL:
   #_w1 := NOT "SS Limit 1 Tranfer1" AND NOT "SS Limit 2 Tranfer1" AND "Edge_164";   // falling edge of "SS Limit 2 Tranfer1"
   "Edge_164" := "SS Limit 2 Tranfer1";
   "TF1_Position_2" := #_w1 OR ("TF1_Position_2" AND NOT "SS Limit 1 Tranfer1");
   #_w2 := "SS Limit 1 Tranfer1" AND NOT "Edge_165";   // rising edge of "SS Limit 1 Tranfer1"
   "Edge_165" := "SS Limit 1 Tranfer1";
   "TF1_Position_1" := (#_w2 AND "SS Limit 2 Tranfer1") OR ("TF1_Position_1" AND "SS Limit 1 Tranfer1");
   #_w3 := NOT "SS Limit 1 Tranfer2" AND NOT "SS Limit 2 Tranfer2" AND "Edge_166";   // falling edge of "SS Limit 2 Tranfer2"
   "Edge_166" := "SS Limit 2 Tranfer2";
   "TF2_Position_2" := (#_w3 AND NOT "SS Limit 3 Tranfer2") OR ("TF2_Position_2" AND "SS Limit 3 Tranfer2" AND NOT "TF2_Position_3");
   "TF2_Position_1" := ("SS Limit 1 Tranfer2" AND "SS Limit 2 Tranfer2" AND "SS Limit 3 Tranfer2") OR "TF2_Position_1";
   "TF2_Position_3" := "SS Limit 2 Tranfer2" AND NOT "SS Limit 3 Tranfer2" AND NOT "SS Limit 1 Tranfer2";
END_REGION

REGION Network 8: XyLanh Control
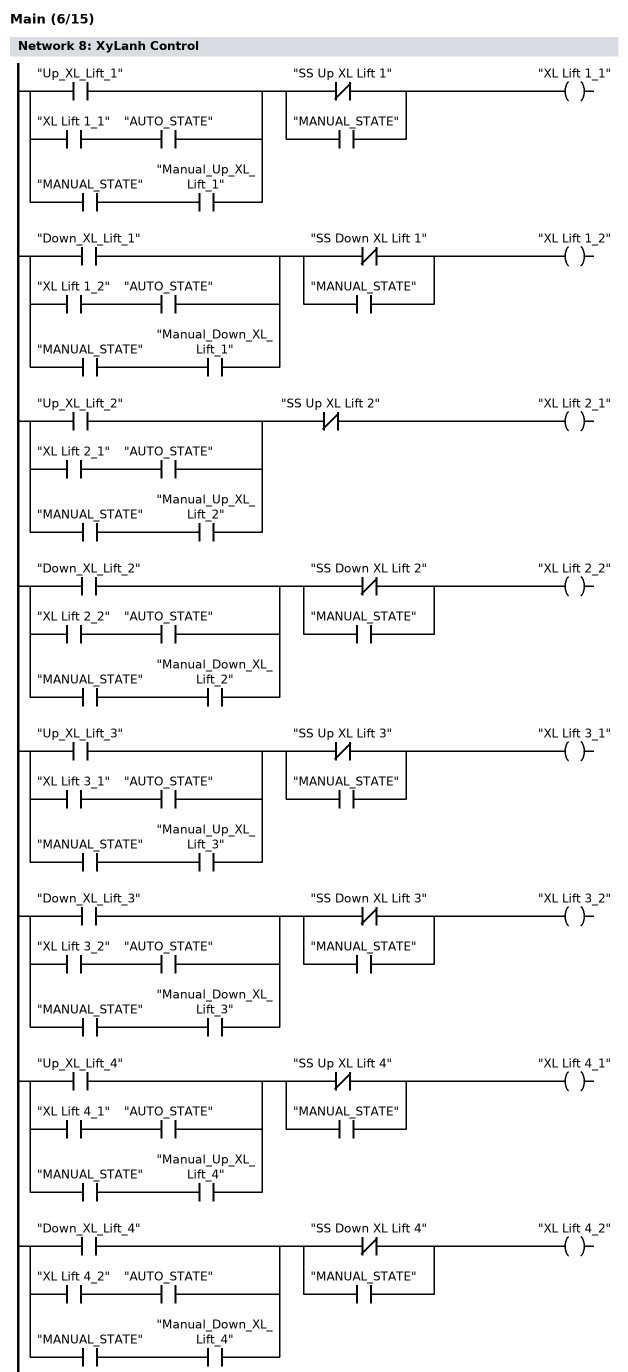
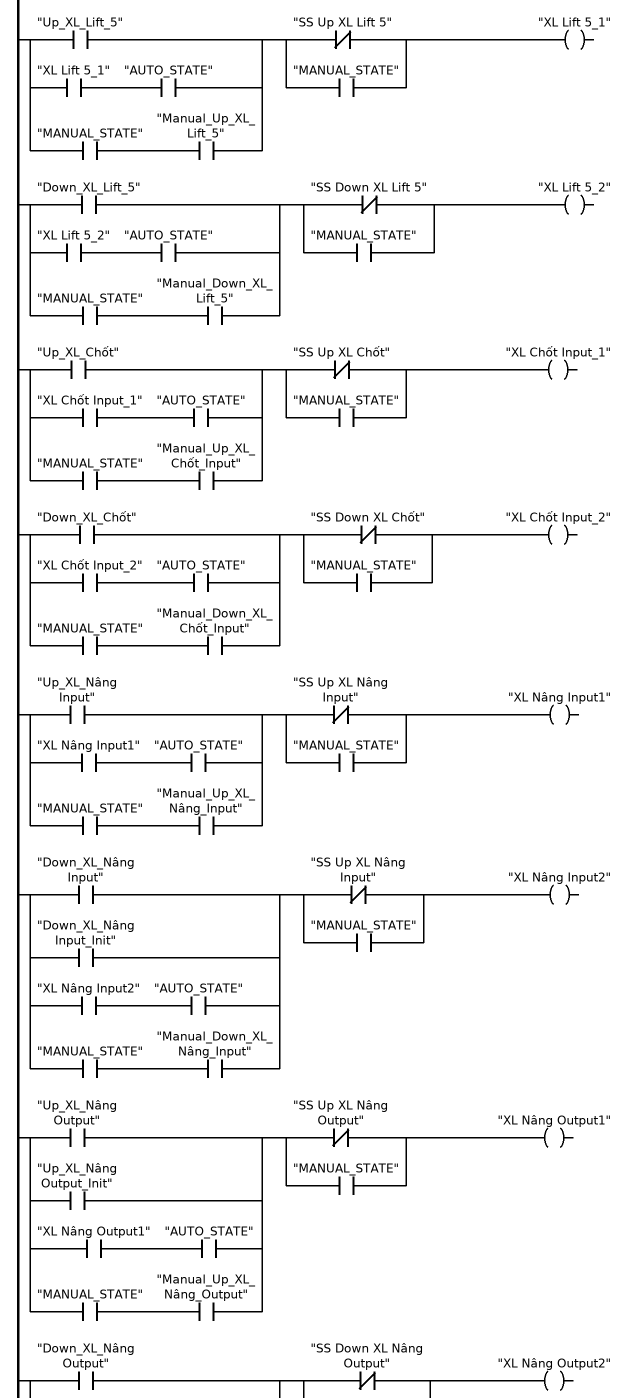
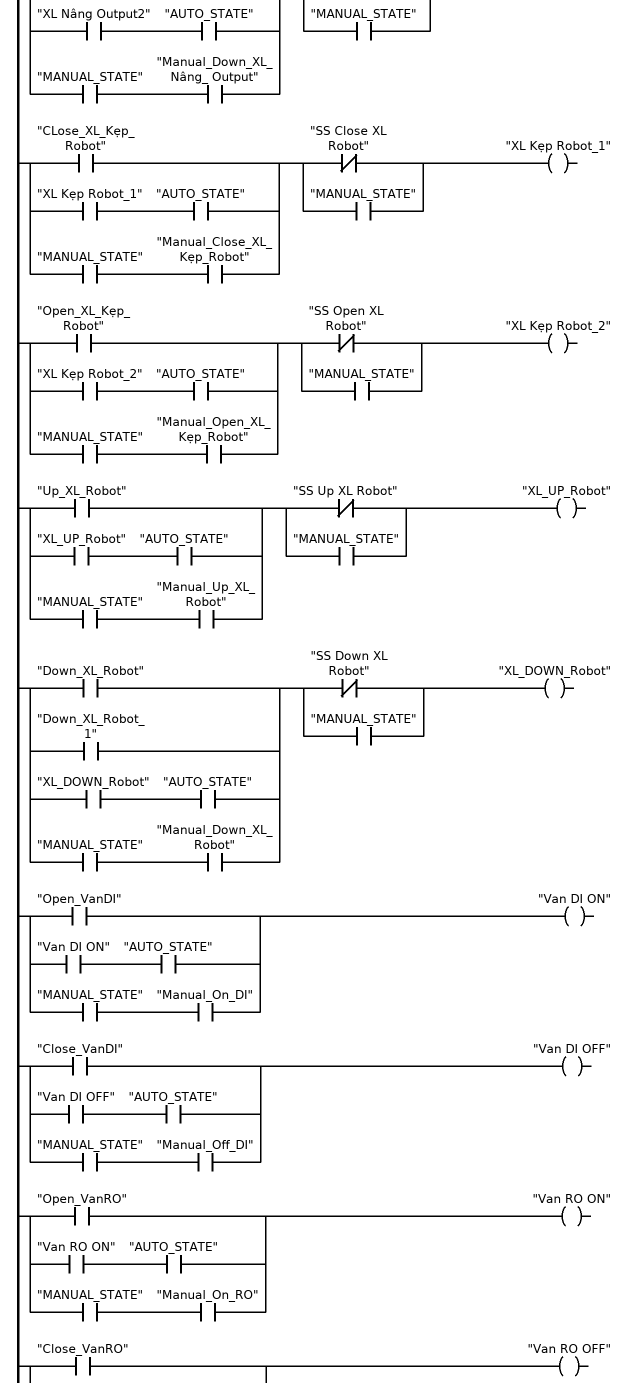
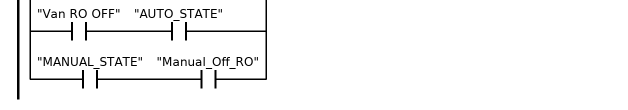
   RUNG wire#powerrail
      Contact( "Up_XL_Lift_1" )
      wire#w1
      I_Contact( "SS Up XL Lift 1" )
      wire#w2
      Coil( "XL Lift 1_1" )
   END_RUNG
   RUNG wire#powerrail
      Contact( "XL Lift 1_1" )
      Contact( "AUTO_STATE" )
   END_RUNG wire#w1
   RUNG wire#powerrail
      Contact( "MANUAL_STATE" )
      Contact( "Manual_Up_XL_Lift_1" )
   END_RUNG wire#w1
   RUNG wire#w1
      Contact( "MANUAL_STATE" )
   END_RUNG wire#w2
   RUNG wire#powerrail
      Contact( "Down_XL_Lift_1" )
      wire#w3
      I_Contact( "SS Down XL Lift 1" )
      wire#w4
      Coil( "XL Lift 1_2" )
   END_RUNG
   RUNG wire#powerrail
      Contact( "XL Lift 1_2" )
      Contact( "AUTO_STATE" )
   END_RUNG wire#w3
   RUNG wire#powerrail
      Contact( "MANUAL_STATE" )
      Contact( "Manual_Down_XL_Lift_1" )
   END_RUNG wire#w3
   RUNG wire#w3
      Contact( "MANUAL_STATE" )
   END_RUNG wire#w4
   RUNG wire#powerrail
      Contact( "Up_XL_Lift_2" )
      wire#w5
      I_Contact( "SS Up XL Lift 2" )
      Coil( "XL Lift 2_1" )
   END_RUNG
   RUNG wire#powerrail
      Contact( "XL Lift 2_1" )
      Contact( "AUTO_STATE" )
   END_RUNG wire#w5
   RUNG wire#powerrail
      Contact( "MANUAL_STATE" )
      Contact( "Manual_Up_XL_Lift_2" )
   END_RUNG wire#w5
   RUNG wire#powerrail
      Contact( "Down_XL_Lift_2" )
      wire#w6
      I_Contact( "SS Down XL Lift 2" )
      wire#w7
      Coil( "XL Lift 2_2" )
   END_RUNG
   RUNG wire#powerrail
      Contact( "XL Lift 2_2" )
      Contact( "AUTO_STATE" )
   END_RUNG wire#w6
   RUNG wire#powerrail
      Contact( "MANUAL_STATE" )
      Contact( "Manual_Down_XL_Lift_2" )
   END_RUNG wire#w6
   RUNG wire#w6
      Contact( "MANUAL_STATE" )
   END_RUNG wire#w7
   RUNG wire#powerrail
      Contact( "Up_XL_Lift_3" )
      wire#w8
      I_Contact( "SS Up XL Lift 3" )
      wire#w9
      Coil( "XL Lift 3_1" )
   END_RUNG
   RUNG wire#powerrail
      Contact( "XL Lift 3_1" )
      Contact( "AUTO_STATE" )
   END_RUNG wire#w8
   RUNG wire#powerrail
      Contact( "MANUAL_STATE" )
      Contact( "Manual_Up_XL_Lift_3" )
   END_RUNG wire#w8
   RUNG wire#w8
      Contact( "MANUAL_STATE" )
   END_RUNG wire#w9
   RUNG wire#powerrail
      Contact( "Down_XL_Lift_3" )
      wire#w10
      I_Contact( "SS Down XL Lift 3" )
      wire#w11
      Coil( "XL Lift 3_2" )
   END_RUNG
   RUNG wire#powerrail
      Contact( "XL Lift 3_2" )
      Contact( "AUTO_STATE" )
   END_RUNG wire#w10
   RUNG wire#powerrail
      Contact( "MANUAL_STATE" )
      Contact( "Manual_Down_XL_Lift_3" )
   END_RUNG wire#w10
   RUNG wire#w10
      Contact( "MANUAL_STATE" )
   END_RUNG wire#w11
   RUNG wire#powerrail
      Contact( "Up_XL_Lift_4" )
      wire#w12
      I_Contact( "SS Up XL Lift 4" )
      wire#w13
      Coil( "XL Lift 4_1" )
   END_RUNG
   RUNG wire#powerrail
      Contact( "XL Lift 4_1" )
      Contact( "AUTO_STATE" )
   END_RUNG wire#w12
   RUNG wire#powerrail
      Contact( "MANUAL_STATE" )
      Contact( "Manual_Up_XL_Lift_4" )
   END_RUNG wire#w12
   RUNG wire#w12
      Contact( "MANUAL_STATE" )
   END_RUNG wire#w13
   RUNG wire#powerrail
      Contact( "Down_XL_Lift_4" )
      wire#w14
      I_Contact( "SS Down XL Lift 4" )
      wire#w15
      Coil( "XL Lift 4_2" )
   END_RUNG
   RUNG wire#powerrail
      Contact( "XL Lift 4_2" )
      Contact( "AUTO_STATE" )
   END_RUNG wire#w14
   RUNG wire#powerrail
      Contact( "MANUAL_STATE" )
      Contact( "Manual_Down_XL_Lift_4" )
   END_RUNG wire#w14
   RUNG wire#w14
      Contact( "MANUAL_STATE" )
   END_RUNG wire#w15
   RUNG wire#powerrail
      Contact( "Up_XL_Lift_5" )
      wire#w16
      I_Contact( "SS Up XL Lift 5" )
      wire#w17
      Coil( "XL Lift 5_1" )
   END_RUNG
   RUNG wire#powerrail
      Contact( "XL Lift 5_1" )
      Contact( "AUTO_STATE" )
   END_RUNG wire#w16
   RUNG wire#powerrail
      Contact( "MANUAL_STATE" )
      Contact( "Manual_Up_XL_Lift_5" )
   END_RUNG wire#w16
   RUNG wire#w16
      Contact( "MANUAL_STATE" )
   END_RUNG wire#w17
   RUNG wire#powerrail
      Contact( "Down_XL_Lift_5" )
      wire#w18
      I_Contact( "SS Down XL Lift 5" )
      wire#w19
      Coil( "XL Lift 5_2" )
   END_RUNG
   RUNG wire#powerrail
      Contact( "XL Lift 5_2" )
      Contact( "AUTO_STATE" )
   END_RUNG wire#w18
   RUNG wire#powerrail
      Contact( "MANUAL_STATE" )
      Contact( "Manual_Down_XL_Lift_5" )
   END_RUNG wire#w18
   RUNG wire#w18
      Contact( "MANUAL_STATE" )
   END_RUNG wire#w19
   RUNG wire#powerrail
      Contact( "Up_XL_Chốt" )
      wire#w20
      I_Contact( "SS Up XL Chốt" )
      wire#w21
      Coil( "XL Chốt Input_1" )
   END_RUNG
   RUNG wire#powerrail
      Contact( "XL Chốt Input_1" )
      Contact( "AUTO_STATE" )
   END_RUNG wire#w20
   RUNG wire#powerrail
      Contact( "MANUAL_STATE" )
      Contact( "Manual_Up_XL_Chốt_Input" )
   END_RUNG wire#w20
   RUNG wire#w20
      Contact( "MANUAL_STATE" )
   END_RUNG wire#w21
   RUNG wire#powerrail
      Contact( "Down_XL_Chốt" )
      wire#w22
      I_Contact( "SS Down XL Chốt" )
      wire#w23
      Coil( "XL Chốt Input_2" )
   END_RUNG
   RUNG wire#powerrail
      Contact( "XL Chốt Input_2" )
      Contact( "AUTO_STATE" )
   END_RUNG wire#w22
   RUNG wire#powerrail
      Contact( "MANUAL_STATE" )
      Contact( "Manual_Down_XL_Chốt_Input" )
   END_RUNG wire#w22
   RUNG wire#w22
      Contact( "MANUAL_STATE" )
   END_RUNG wire#w23
   RUNG wire#powerrail
      Contact( "Up_XL_Nâng Input" )
      wire#w24
      I_Contact( "SS Up XL Nâng Input" )
      wire#w25
      Coil( "XL Nâng Input1" )
   END_RUNG
   RUNG wire#powerrail
      Contact( "XL Nâng Input1" )
      Contact( "AUTO_STATE" )
   END_RUNG wire#w24
   RUNG wire#powerrail
      Contact( "MANUAL_STATE" )
      Contact( "Manual_Up_XL_Nâng_Input" )
   END_RUNG wire#w24
   RUNG wire#w24
      Contact( "MANUAL_STATE" )
   END_RUNG wire#w25
   RUNG wire#powerrail
      Contact( "Down_XL_Nâng Input" )
      wire#w26
      I_Contact( "SS Up XL Nâng Input" )
      wire#w27
      Coil( "XL Nâng Input2" )
   END_RUNG
   RUNG wire#powerrail
      Contact( "Down_XL_Nâng Input_Init" )
   END_RUNG wire#w26
   RUNG wire#powerrail
      Contact( "XL Nâng Input2" )
      Contact( "AUTO_STATE" )
   END_RUNG wire#w26
   RUNG wire#powerrail
      Contact( "MANUAL_STATE" )
      Contact( "Manual_Down_XL_Nâng_Input" )
   END_RUNG wire#w26
   RUNG wire#w26
      Contact( "MANUAL_STATE" )
   END_RUNG wire#w27
   RUNG wire#powerrail
      Contact( "Up_XL_Nâng Output" )
      wire#w28
      I_Contact( "SS Up XL Nâng Output" )
      wire#w29
      Coil( "XL Nâng Output1" )
   END_RUNG
   RUNG wire#powerrail
      Contact( "Up_XL_Nâng Output_Init" )
   END_RUNG wire#w28
   RUNG wire#powerrail
      Contact( "XL Nâng Output1" )
      Contact( "AUTO_STATE" )
   END_RUNG wire#w28
   RUNG wire#powerrail
      Contact( "MANUAL_STATE" )
      Contact( "Manual_Up_XL_Nâng_Output" )
   END_RUNG wire#w28
   RUNG wire#w28
      Contact( "MANUAL_STATE" )
   END_RUNG wire#w29
   RUNG wire#powerrail
      Contact( "Down_XL_Nâng Output" )
      wire#w30
      I_Contact( "SS Down XL Nâng Output" )
      wire#w31
      Coil( "XL Nâng Output2" )
   END_RUNG
   RUNG wire#powerrail
      Contact( "XL Nâng Output2" )
      Contact( "AUTO_STATE" )
   END_RUNG wire#w30
   RUNG wire#powerrail
      Contact( "MANUAL_STATE" )
      Contact( "Manual_Down_XL_Nâng_ Output" )
   END_RUNG wire#w30
   RUNG wire#w30
      Contact( "MANUAL_STATE" )
   END_RUNG wire#w31
   RUNG wire#powerrail
      Contact( "CLose_XL_Kẹp_Robot" )
      wire#w32
      I_Contact( "SS Close XL Robot" )
      wire#w33
      Coil( "XL Kẹp Robot_1" )
   END_RUNG
   RUNG wire#powerrail
      Contact( "XL Kẹp Robot_1" )
      Contact( "AUTO_STATE" )
   END_RUNG wire#w32
   RUNG wire#powerrail
      Contact( "MANUAL_STATE" )
      Contact( "Manual_Close_XL_Kẹp_Robot" )
   END_RUNG wire#w32
   RUNG wire#w32
      Contact( "MANUAL_STATE" )
   END_RUNG wire#w33
   RUNG wire#powerrail
      Contact( "Open_XL_Kẹp_Robot" )
      wire#w34
      I_Contact( "SS Open XL Robot" )
      wire#w35
      Coil( "XL Kẹp Robot_2" )
   END_RUNG
   RUNG wire#powerrail
      Contact( "XL Kẹp Robot_2" )
      Contact( "AUTO_STATE" )
   END_RUNG wire#w34
   RUNG wire#powerrail
      Contact( "MANUAL_STATE" )
      Contact( "Manual_Open_XL_Kẹp_Robot" )
   END_RUNG wire#w34
   RUNG wire#w34
      Contact( "MANUAL_STATE" )
   END_RUNG wire#w35
   RUNG wire#powerrail
      Contact( "Up_XL_Robot" )
      wire#w36
      I_Contact( "SS Up XL Robot" )
      wire#w37
      Coil( "XL_UP_Robot" )
   END_RUNG
   RUNG wire#powerrail
      Contact( "XL_UP_Robot" )
      Contact( "AUTO_STATE" )
   END_RUNG wire#w36
   RUNG wire#powerrail
      Contact( "MANUAL_STATE" )
      Contact( "Manual_Up_XL_Robot" )
   END_RUNG wire#w36
   RUNG wire#w36
      Contact( "MANUAL_STATE" )
   END_RUNG wire#w37
   RUNG wire#powerrail
      Contact( "Down_XL_Robot" )
      wire#w38
      I_Contact( "SS Down XL Robot" )
      wire#w39
      Coil( "XL_DOWN_Robot" )
   END_RUNG
   RUNG wire#powerrail
      Contact( "Down_XL_Robot_1" )
   END_RUNG wire#w38
   RUNG wire#powerrail
      Contact( "XL_DOWN_Robot" )
      Contact( "AUTO_STATE" )
   END_RUNG wire#w38
   RUNG wire#powerrail
      Contact( "MANUAL_STATE" )
      Contact( "Manual_Down_XL_Robot" )
   END_RUNG wire#w38
   RUNG wire#w38
      Contact( "MANUAL_STATE" )
   END_RUNG wire#w39
   RUNG wire#powerrail
      Contact( "Open_VanDI" )
      wire#w40
      Coil( "Van DI ON" )
   END_RUNG
   RUNG wire#powerrail
      Contact( "Van DI ON" )
      Contact( "AUTO_STATE" )
   END_RUNG wire#w40
   RUNG wire#powerrail
      Contact( "MANUAL_STATE" )
      Contact( "Manual_On_DI" )
   END_RUNG wire#w40
   RUNG wire#powerrail
      Contact( "Close_VanDI" )
      wire#w41
      Coil( "Van DI OFF" )
   END_RUNG
   RUNG wire#powerrail
      Contact( "Van DI OFF" )
      Contact( "AUTO_STATE" )
   END_RUNG wire#w41
   RUNG wire#powerrail
      Contact( "MANUAL_STATE" )
      Contact( "Manual_Off_DI" )
   END_RUNG wire#w41
   RUNG wire#powerrail
      Contact( "Open_VanRO" )
      wire#w42
      Coil( "Van RO ON" )
   END_RUNG
   RUNG wire#powerrail
      Contact( "Van RO ON" )
      Contact( "AUTO_STATE" )
   END_RUNG wire#w42
   RUNG wire#powerrail
      Contact( "MANUAL_STATE" )
      Contact( "Manual_On_RO" )
   END_RUNG wire#w42
   RUNG wire#powerrail
      Contact( "Close_VanRO" )
      wire#w43
      Coil( "Van RO OFF" )
   END_RUNG
   RUNG wire#powerrail
      Contact( "Van RO OFF" )
      Contact( "AUTO_STATE" )
   END_RUNG wire#w43
   RUNG wire#powerrail
      Contact( "MANUAL_STATE" )
      Contact( "Manual_Off_RO" )
   END_RUNG wire#w43
   // the same network as SCL:
   "XL Lift 1_1" := ("Up_XL_Lift_1" OR ("XL Lift 1_1" AND "AUTO_STATE") OR ("MANUAL_STATE" AND "Manual_Up_XL_Lift_1")) AND (NOT "SS Up XL Lift 1" OR "MANUAL_STATE");
   "XL Lift 1_2" := ("Down_XL_Lift_1" OR ("XL Lift 1_2" AND "AUTO_STATE") OR ("MANUAL_STATE" AND "Manual_Down_XL_Lift_1")) AND (NOT "SS Down XL Lift 1" OR "MANUAL_STATE");
   "XL Lift 2_1" := ("Up_XL_Lift_2" OR ("XL Lift 2_1" AND "AUTO_STATE") OR ("MANUAL_STATE" AND "Manual_Up_XL_Lift_2")) AND NOT "SS Up XL Lift 2";
   "XL Lift 2_2" := ("Down_XL_Lift_2" OR ("XL Lift 2_2" AND "AUTO_STATE") OR ("MANUAL_STATE" AND "Manual_Down_XL_Lift_2")) AND (NOT "SS Down XL Lift 2" OR "MANUAL_STATE");
   "XL Lift 3_1" := ("Up_XL_Lift_3" OR ("XL Lift 3_1" AND "AUTO_STATE") OR ("MANUAL_STATE" AND "Manual_Up_XL_Lift_3")) AND (NOT "SS Up XL Lift 3" OR "MANUAL_STATE");
   "XL Lift 3_2" := ("Down_XL_Lift_3" OR ("XL Lift 3_2" AND "AUTO_STATE") OR ("MANUAL_STATE" AND "Manual_Down_XL_Lift_3")) AND (NOT "SS Down XL Lift 3" OR "MANUAL_STATE");
   "XL Lift 4_1" := ("Up_XL_Lift_4" OR ("XL Lift 4_1" AND "AUTO_STATE") OR ("MANUAL_STATE" AND "Manual_Up_XL_Lift_4")) AND (NOT "SS Up XL Lift 4" OR "MANUAL_STATE");
   "XL Lift 4_2" := ("Down_XL_Lift_4" OR ("XL Lift 4_2" AND "AUTO_STATE") OR ("MANUAL_STATE" AND "Manual_Down_XL_Lift_4")) AND (NOT "SS Down XL Lift 4" OR "MANUAL_STATE");
   "XL Lift 5_1" := ("Up_XL_Lift_5" OR ("XL Lift 5_1" AND "AUTO_STATE") OR ("MANUAL_STATE" AND "Manual_Up_XL_Lift_5")) AND (NOT "SS Up XL Lift 5" OR "MANUAL_STATE");
   "XL Lift 5_2" := ("Down_XL_Lift_5" OR ("XL Lift 5_2" AND "AUTO_STATE") OR ("MANUAL_STATE" AND "Manual_Down_XL_Lift_5")) AND (NOT "SS Down XL Lift 5" OR "MANUAL_STATE");
   "XL Chốt Input_1" := ("Up_XL_Chốt" OR ("XL Chốt Input_1" AND "AUTO_STATE") OR ("MANUAL_STATE" AND "Manual_Up_XL_Chốt_Input")) AND (NOT "SS Up XL Chốt" OR "MANUAL_STATE");
   "XL Chốt Input_2" := ("Down_XL_Chốt" OR ("XL Chốt Input_2" AND "AUTO_STATE") OR ("MANUAL_STATE" AND "Manual_Down_XL_Chốt_Input")) AND (NOT "SS Down XL Chốt" OR "MANUAL_STATE");
   "XL Nâng Input1" := ("Up_XL_Nâng Input" OR ("XL Nâng Input1" AND "AUTO_STATE") OR ("MANUAL_STATE" AND "Manual_Up_XL_Nâng_Input")) AND (NOT "SS Up XL Nâng Input" OR "MANUAL_STATE");
   "XL Nâng Input2" := ("Down_XL_Nâng Input" OR "Down_XL_Nâng Input_Init" OR ("XL Nâng Input2" AND "AUTO_STATE") OR ("MANUAL_STATE" AND "Manual_Down_XL_Nâng_Input")) AND (NOT "SS Up XL Nâng Input" OR "MANUAL_STATE");
   "XL Nâng Output1" := ("Up_XL_Nâng Output" OR "Up_XL_Nâng Output_Init" OR ("XL Nâng Output1" AND "AUTO_STATE") OR ("MANUAL_STATE" AND "Manual_Up_XL_Nâng_Output")) AND (NOT "SS Up XL Nâng Output" OR "MANUAL_STATE");
   "XL Nâng Output2" := ("Down_XL_Nâng Output" OR ("XL Nâng Output2" AND "AUTO_STATE") OR ("MANUAL_STATE" AND "Manual_Down_XL_Nâng_ Output")) AND (NOT "SS Down XL Nâng Output" OR "MANUAL_STATE");
   "XL Kẹp Robot_1" := ("CLose_XL_Kẹp_Robot" OR ("XL Kẹp Robot_1" AND "AUTO_STATE") OR ("MANUAL_STATE" AND "Manual_Close_XL_Kẹp_Robot")) AND (NOT "SS Close XL Robot" OR "MANUAL_STATE");
   "XL Kẹp Robot_2" := ("Open_XL_Kẹp_Robot" OR ("XL Kẹp Robot_2" AND "AUTO_STATE") OR ("MANUAL_STATE" AND "Manual_Open_XL_Kẹp_Robot")) AND (NOT "SS Open XL Robot" OR "MANUAL_STATE");
   "XL_UP_Robot" := ("Up_XL_Robot" OR ("XL_UP_Robot" AND "AUTO_STATE") OR ("MANUAL_STATE" AND "Manual_Up_XL_Robot")) AND (NOT "SS Up XL Robot" OR "MANUAL_STATE");
   "XL_DOWN_Robot" := ("Down_XL_Robot" OR "Down_XL_Robot_1" OR ("XL_DOWN_Robot" AND "AUTO_STATE") OR ("MANUAL_STATE" AND "Manual_Down_XL_Robot")) AND (NOT "SS Down XL Robot" OR "MANUAL_STATE");
   "Van DI ON" := "Open_VanDI" OR ("Van DI ON" AND "AUTO_STATE") OR ("MANUAL_STATE" AND "Manual_On_DI");
   "Van DI OFF" := "Close_VanDI" OR ("Van DI OFF" AND "AUTO_STATE") OR ("MANUAL_STATE" AND "Manual_Off_DI");
   "Van RO ON" := "Open_VanRO" OR ("Van RO ON" AND "AUTO_STATE") OR ("MANUAL_STATE" AND "Manual_On_RO");
   "Van RO OFF" := "Close_VanRO" OR ("Van RO OFF" AND "AUTO_STATE") OR ("MANUAL_STATE" AND "Manual_Off_RO");
END_REGION

REGION Network 9: Begin Precess
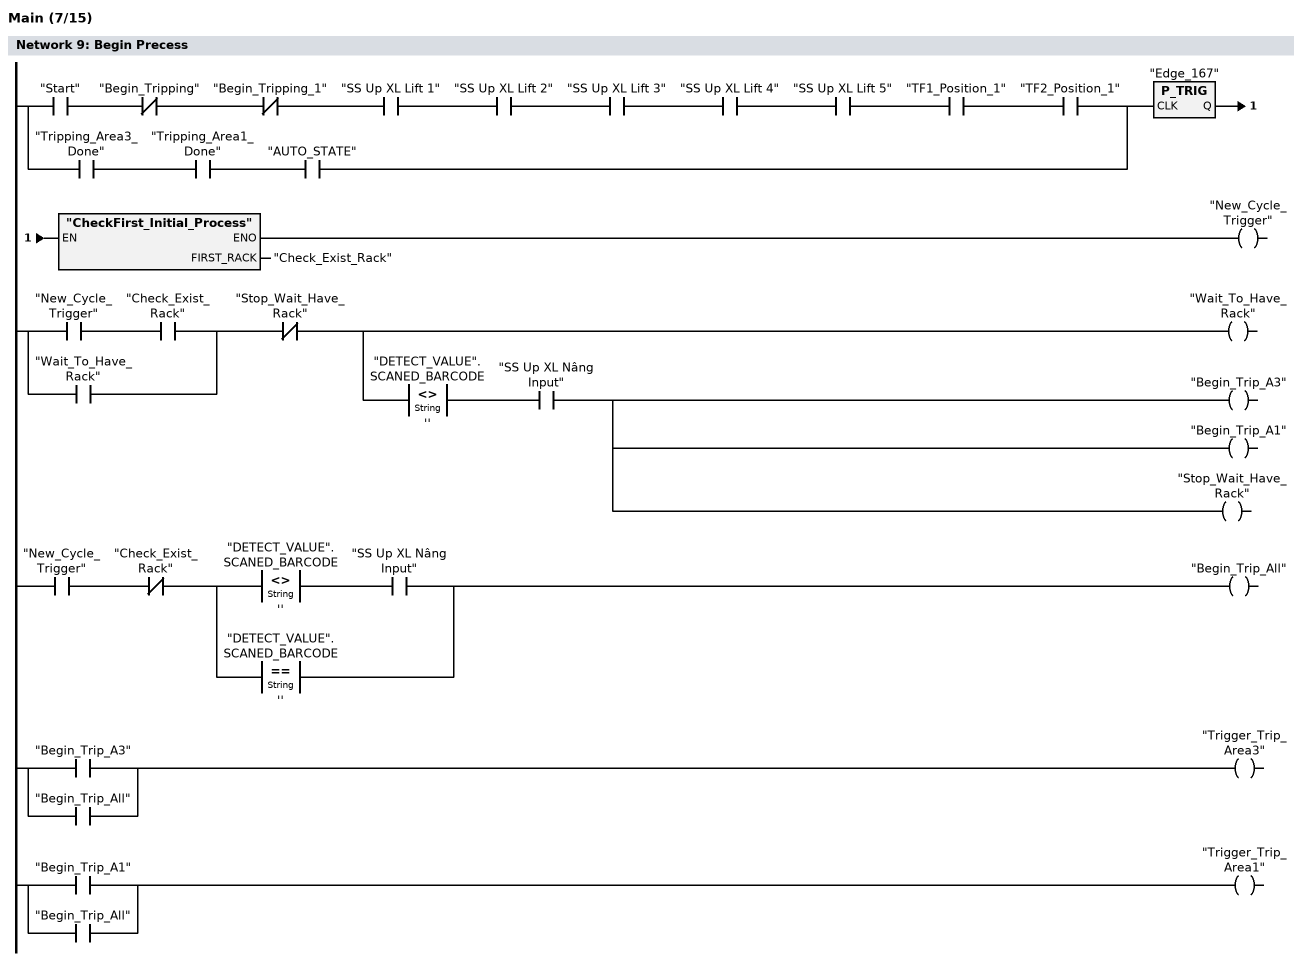
   RUNG wire#powerrail
      Contact( "Start" )
      I_Contact( "Begin_Tripping" )
      I_Contact( "Begin_Tripping_1" )
      Contact( "SS Up XL Lift 1" )
      Contact( "SS Up XL Lift 2" )
      Contact( "SS Up XL Lift 3" )
      Contact( "SS Up XL Lift 4" )
      Contact( "SS Up XL Lift 5" )
      Contact( "TF1_Position_1" )
      Contact( "TF2_Position_1" )
      wire#w1
      P_Trig( "Edge_167" )
      "CheckFirst_Initial_Process"(FIRST_RACK => "Check_Exist_Rack")
      Coil( "New_Cycle_Trigger" )
   END_RUNG
   RUNG wire#powerrail
      Contact( "Tripping_Area3_Done" )
      Contact( "Tripping_Area1_Done" )
      Contact( "AUTO_STATE" )
   END_RUNG wire#w1
   RUNG wire#powerrail
      Contact( "New_Cycle_Trigger" )
      Contact( "Check_Exist_Rack" )
      wire#w2
      I_Contact( "Stop_Wait_Have_Rack" )
      wire#w3
      Coil( "Wait_To_Have_Rack" )
   END_RUNG
   RUNG wire#powerrail
      Contact( "Wait_To_Have_Rack" )
   END_RUNG wire#w2
   RUNG wire#w3
      { S7_Templates := "SrcType := String" } NE_Contact(in1 := "DETECT_VALUE".SCANED_BARCODE, in2 := '')
      Contact( "SS Up XL Nâng Input" )
      wire#w4
      Coil( "Begin_Trip_A3" )
   END_RUNG
   RUNG wire#w4
      Coil( "Begin_Trip_A1" )
   END_RUNG
   RUNG wire#w4
      Coil( "Stop_Wait_Have_Rack" )
   END_RUNG
   RUNG wire#powerrail
      Contact( "New_Cycle_Trigger" )
      I_Contact( "Check_Exist_Rack" )
      wire#w5
      { S7_Templates := "SrcType := String" } NE_Contact(in1 := "DETECT_VALUE".SCANED_BARCODE, in2 := '')
      Contact( "SS Up XL Nâng Input" )
      wire#w6
      Coil( "Begin_Trip_All" )
   END_RUNG
   RUNG wire#w5
      { S7_Templates := "SrcType := String" } EQ_Contact(in1 := "DETECT_VALUE".SCANED_BARCODE, in2 := '')
   END_RUNG wire#w6
   RUNG wire#powerrail
      Contact( "Begin_Trip_A3" )
      wire#w7
      Coil( "Trigger_Trip_Area3" )
   END_RUNG
   RUNG wire#powerrail
      Contact( "Begin_Trip_All" )
   END_RUNG wire#w7
   RUNG wire#powerrail
      Contact( "Begin_Trip_A1" )
      wire#w8
      Coil( "Trigger_Trip_Area1" )
   END_RUNG
   RUNG wire#powerrail
      Contact( "Begin_Trip_All" )
   END_RUNG wire#w8
   // the same network as SCL:
   #_w1 := ("Start" AND NOT "Begin_Tripping" AND NOT "Begin_Tripping_1" AND "SS Up XL Lift 1" AND "SS Up XL Lift 2" AND "SS Up XL Lift 3" AND "SS Up XL Lift 4" AND "SS Up XL Lift 5" AND "TF1_Position_1" AND "TF2_Position_1") OR ("Tripping_Area3_Done" AND "Tripping_Area1_Done" AND "AUTO_STATE");
   #_w2 := #_w1 AND NOT "Edge_167";   // rising edge
   "Edge_167" := #_w1;
   "CheckFirst_Initial_Process"(EN := #_w2, FIRST_RACK => "Check_Exist_Rack", ENO => #_w3);
   "New_Cycle_Trigger" := #_w3;
   "Wait_To_Have_Rack" := (("New_Cycle_Trigger" AND "Check_Exist_Rack") OR "Wait_To_Have_Rack") AND NOT "Stop_Wait_Have_Rack";
   "Begin_Trip_A3" := "Wait_To_Have_Rack" AND ("DETECT_VALUE".SCANED_BARCODE <> '') AND "SS Up XL Nâng Input";
   "Begin_Trip_A1" := "Begin_Trip_A3";
   "Stop_Wait_Have_Rack" := "Begin_Trip_A3";
   "Begin_Trip_All" := "New_Cycle_Trigger" AND NOT "Check_Exist_Rack" AND ((("DETECT_VALUE".SCANED_BARCODE <> '') AND "SS Up XL Nâng Input") OR ("DETECT_VALUE".SCANED_BARCODE = ''));
   "Trigger_Trip_Area3" := "Begin_Trip_A3" OR "Begin_Trip_All";
   "Trigger_Trip_Area1" := "Begin_Trip_A1" OR "Begin_Trip_All";
END_REGION

REGION Network 10: Prepare -> Tripping Area 1
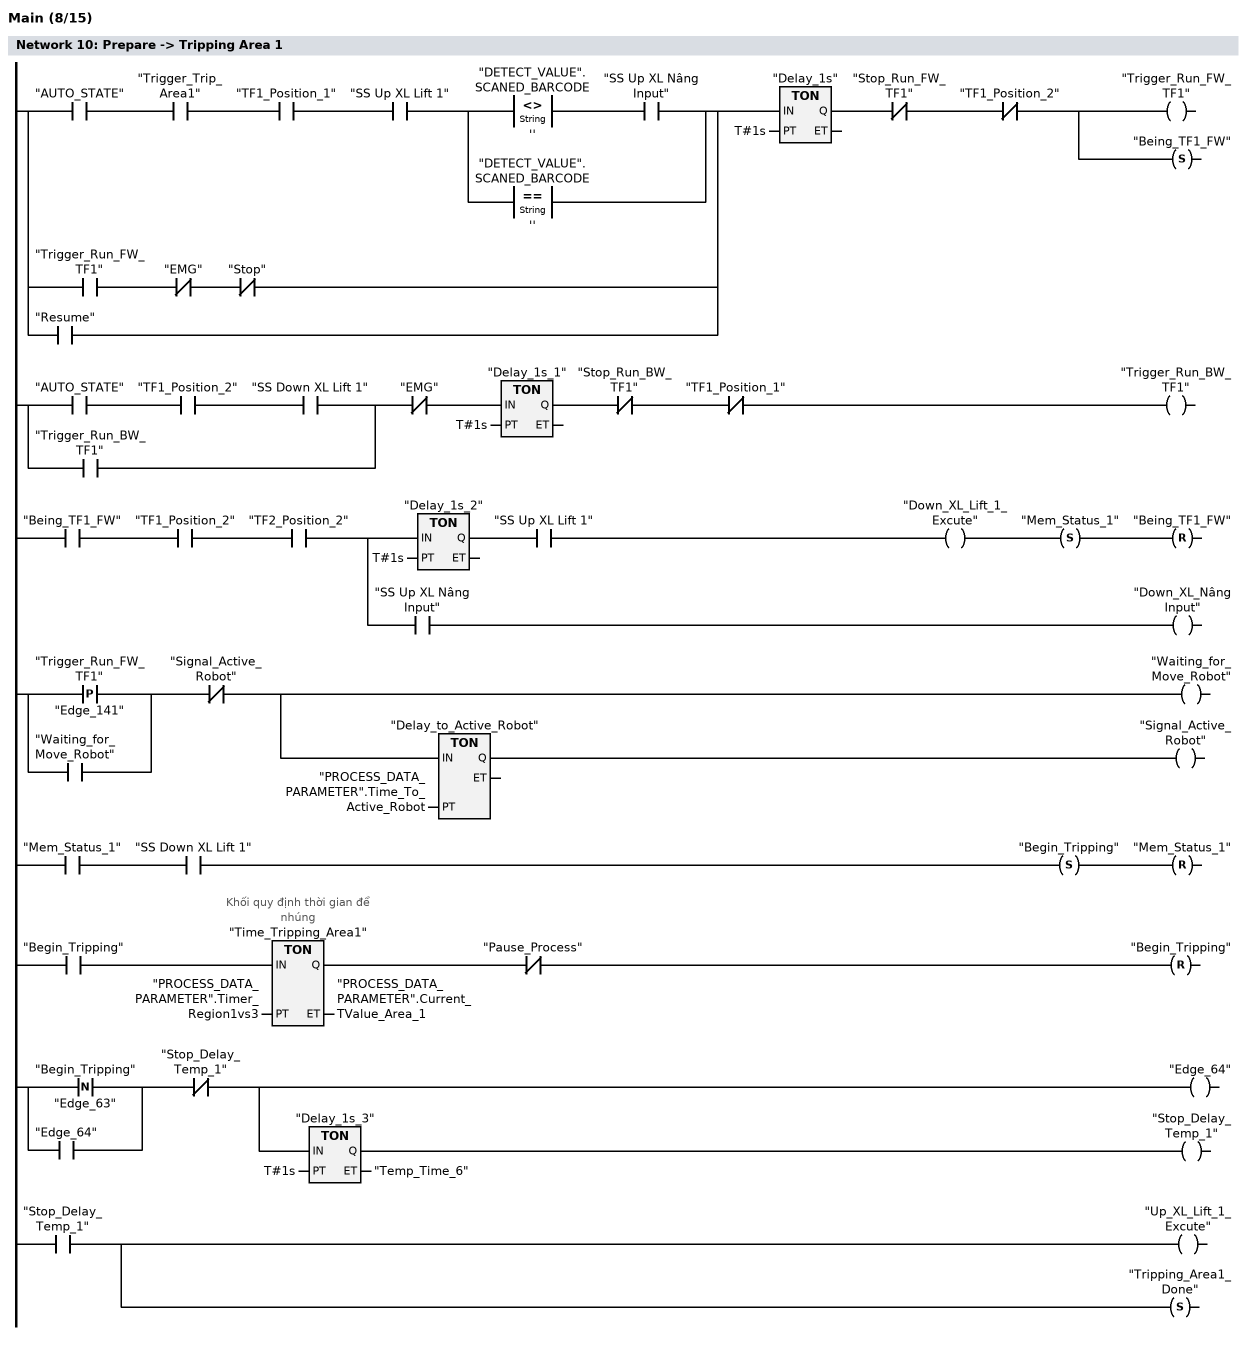
   "Delay_1s".TON(IN := ("AUTO_STATE" AND "Trigger_Trip_Area1" AND "TF1_Position_1" AND "SS Up XL Lift 1" AND ((("DETECT_VALUE".SCANED_BARCODE <> '') AND "SS Up XL Nâng Input") OR ("DETECT_VALUE".SCANED_BARCODE = ''))) OR ("Trigger_Run_FW_TF1" AND NOT "EMG" AND NOT "Stop") OR "Resume",
                  PT := T#1s);
   "Trigger_Run_FW_TF1" := "Delay_1s".Q AND NOT "Stop_Run_FW_TF1" AND NOT "TF1_Position_2";
   IF "Trigger_Run_FW_TF1" THEN "Being_TF1_FW" := TRUE; END_IF;
   "Delay_1s_1".TON(IN := (("AUTO_STATE" AND "TF1_Position_2" AND "SS Down XL Lift 1") OR "Trigger_Run_BW_TF1") AND NOT "EMG",
                    PT := T#1s);
   "Trigger_Run_BW_TF1" := "Delay_1s_1".Q AND NOT "Stop_Run_BW_TF1" AND NOT "TF1_Position_1";
   #_w1 := "Being_TF1_FW" AND "TF1_Position_2" AND "TF2_Position_2";
   "Delay_1s_2".TON(IN := #_w1, PT := T#1s);
   "Down_XL_Lift_1_Excute" := "Delay_1s_2".Q AND "SS Up XL Lift 1";
   IF "Down_XL_Lift_1_Excute" THEN
       "Mem_Status_1" := TRUE;
       "Being_TF1_FW" := FALSE;
   END_IF;
   "Down_XL_Nâng Input" := #_w1 AND "SS Up XL Nâng Input";
   #_w2 := "Trigger_Run_FW_TF1" AND NOT "Edge_141";   // rising edge of "Trigger_Run_FW_TF1"
   "Edge_141" := "Trigger_Run_FW_TF1";
   "Waiting_for_Move_Robot" := (#_w2 OR "Waiting_for_Move_Robot") AND NOT "Signal_Active_Robot";
   "Delay_to_Active_Robot".TON(IN := "Waiting_for_Move_Robot",
                           PT := "PROCESS_DATA_PARAMETER".Time_To_Active_Robot);
   "Signal_Active_Robot" := "Delay_to_Active_Robot".Q;
   IF "Mem_Status_1" AND "SS Down XL Lift 1" THEN
       "Begin_Tripping" := TRUE;
       "Mem_Status_1" := FALSE;
   END_IF;
   "Time_Tripping_Area1".TON(IN := "Begin_Tripping",   // Khối quy định thời gian để nhúng
                           PT := "PROCESS_DATA_PARAMETER".Timer_Region1vs3,
                           ET => "PROCESS_DATA_PARAMETER".Current_TValue_Area_1);
   IF "Time_Tripping_Area1".Q AND NOT "Pause_Process" THEN "Begin_Tripping" := FALSE; END_IF;
   #_w3 := NOT "Begin_Tripping" AND "Edge_63";   // falling edge of "Begin_Tripping"
   "Edge_63" := "Begin_Tripping";
   "Edge_64" := (#_w3 OR "Edge_64") AND NOT "Stop_Delay_Temp_1";
   "Delay_1s_3".TON(IN := "Edge_64", PT := T#1s, ET => "Temp_Time_6");
   "Stop_Delay_Temp_1" := "Delay_1s_3".Q;
   "Up_XL_Lift_1_Excute" := "Stop_Delay_Temp_1";
   IF "Stop_Delay_Temp_1" THEN "Tripping_Area1_Done" := TRUE; END_IF;
END_REGION

REGION Network 11: Trigger Run Lift 1 FW
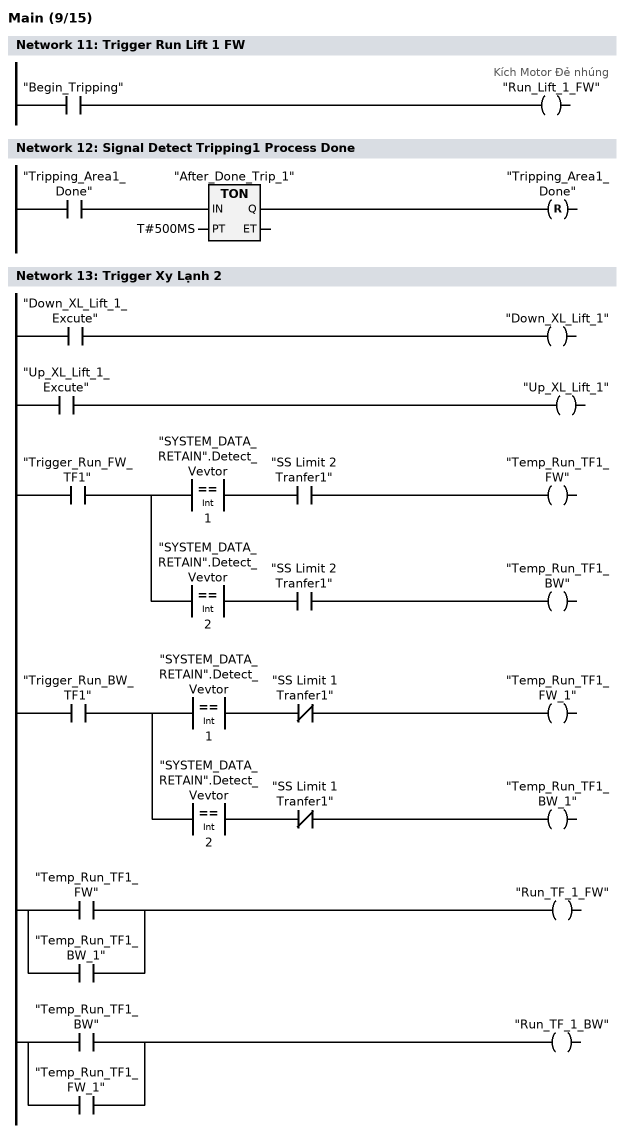
   RUNG wire#powerrail
      Contact( "Begin_Tripping" )
      Coil( "Run_Lift_1_FW" )   // Kích Motor Đẻ nhúng
   END_RUNG
   // the same network as SCL:
   "Run_Lift_1_FW" := "Begin_Tripping";   // Kích Motor Đẻ nhúng
END_REGION

REGION Network 12: Signal Detect Tripping1 Process Done
   "After_Done_Trip_1".TON(IN := "Tripping_Area1_Done", PT := T#500MS);
   IF "After_Done_Trip_1".Q THEN "Tripping_Area1_Done" := FALSE; END_IF;
END_REGION

REGION Network 13: Trigger Xy Lạnh 2
   RUNG wire#powerrail
      Contact( "Down_XL_Lift_1_Excute" )
      Coil( "Down_XL_Lift_1" )
   END_RUNG
   RUNG wire#powerrail
      Contact( "Up_XL_Lift_1_Excute" )
      Coil( "Up_XL_Lift_1" )
   END_RUNG
   RUNG wire#powerrail
      Contact( "Trigger_Run_FW_TF1" )
      wire#w1
      { S7_Templates := "SrcType := Int" } EQ_Contact(in1 := "SYSTEM_DATA_RETAIN".Detect_Vevtor, in2 := 1)
      Contact( "SS Limit 2 Tranfer1" )
      Coil( "Temp_Run_TF1_FW" )
   END_RUNG
   RUNG wire#w1
      { S7_Templates := "SrcType := Int" } EQ_Contact(in1 := "SYSTEM_DATA_RETAIN".Detect_Vevtor, in2 := 2)
      Contact( "SS Limit 2 Tranfer1" )
      Coil( "Temp_Run_TF1_BW" )
   END_RUNG
   RUNG wire#powerrail
      Contact( "Trigger_Run_BW_TF1" )
      wire#w2
      { S7_Templates := "SrcType := Int" } EQ_Contact(in1 := "SYSTEM_DATA_RETAIN".Detect_Vevtor, in2 := 1)
      I_Contact( "SS Limit 1 Tranfer1" )
      Coil( "Temp_Run_TF1_FW_1" )
   END_RUNG
   RUNG wire#w2
      { S7_Templates := "SrcType := Int" } EQ_Contact(in1 := "SYSTEM_DATA_RETAIN".Detect_Vevtor, in2 := 2)
      I_Contact( "SS Limit 1 Tranfer1" )
      Coil( "Temp_Run_TF1_BW_1" )
   END_RUNG
   RUNG wire#powerrail
      Contact( "Temp_Run_TF1_FW" )
      wire#w3
      Coil( "Run_TF_1_FW" )
   END_RUNG
   RUNG wire#powerrail
      Contact( "Temp_Run_TF1_BW_1" )
   END_RUNG wire#w3
   RUNG wire#powerrail
      Contact( "Temp_Run_TF1_BW" )
      wire#w4
      Coil( "Run_TF_1_BW" )
   END_RUNG
   RUNG wire#powerrail
      Contact( "Temp_Run_TF1_FW_1" )
   END_RUNG wire#w4
   // the same network as SCL:
   "Down_XL_Lift_1" := "Down_XL_Lift_1_Excute";
   "Up_XL_Lift_1" := "Up_XL_Lift_1_Excute";
   "Temp_Run_TF1_FW" := "Trigger_Run_FW_TF1" AND ("SYSTEM_DATA_RETAIN".Detect_Vevtor = 1) AND "SS Limit 2 Tranfer1";
   "Temp_Run_TF1_BW" := "Trigger_Run_FW_TF1" AND ("SYSTEM_DATA_RETAIN".Detect_Vevtor = 2) AND "SS Limit 2 Tranfer1";
   "Temp_Run_TF1_FW_1" := "Trigger_Run_BW_TF1" AND ("SYSTEM_DATA_RETAIN".Detect_Vevtor = 1) AND NOT "SS Limit 1 Tranfer1";
   "Temp_Run_TF1_BW_1" := "Trigger_Run_BW_TF1" AND ("SYSTEM_DATA_RETAIN".Detect_Vevtor = 2) AND NOT "SS Limit 1 Tranfer1";
   "Run_TF_1_FW" := "Temp_Run_TF1_FW" OR "Temp_Run_TF1_BW_1";
   "Run_TF_1_BW" := "Temp_Run_TF1_BW" OR "Temp_Run_TF1_FW_1";
END_REGION

REGION Network 14: Prepare -> Tripping Area 3
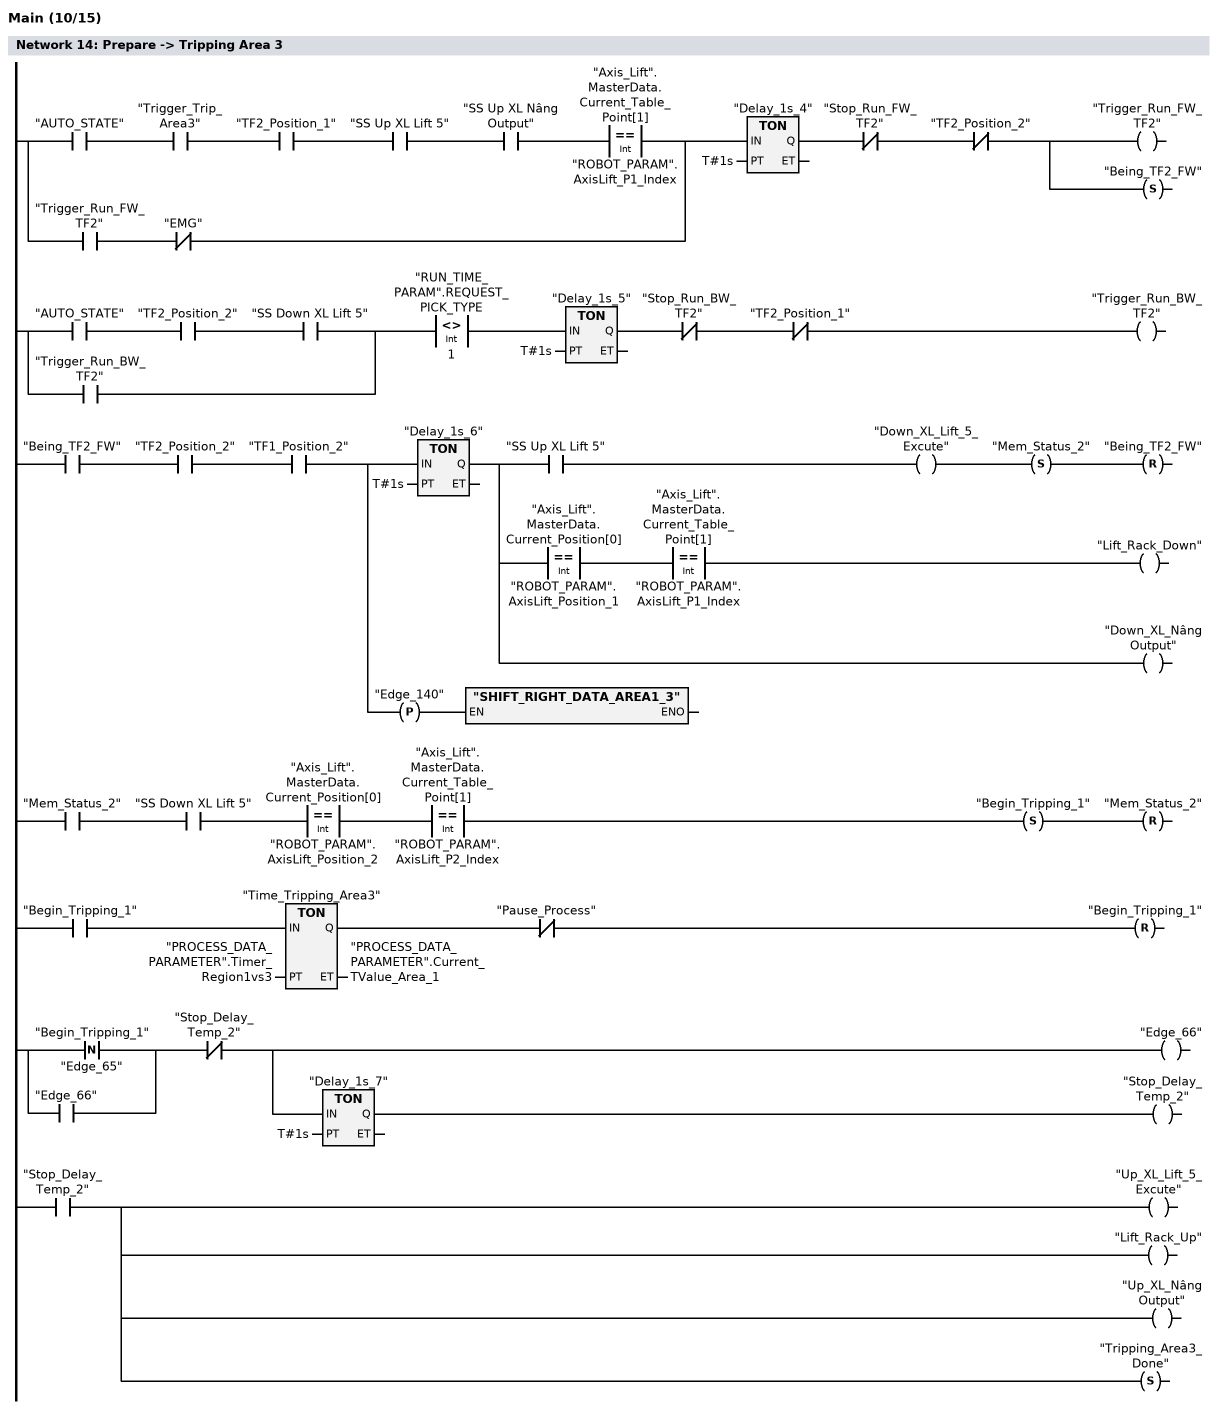
   "Delay_1s_4".TON(IN := ("AUTO_STATE" AND "Trigger_Trip_Area3" AND "TF2_Position_1" AND "SS Up XL Lift 5" AND "SS Up XL Nâng Output" AND ("Axis_Lift".MasterData.Current_Table_Point[1] = "ROBOT_PARAM".AxisLift_P1_Index)) OR ("Trigger_Run_FW_TF2" AND NOT "EMG"),
                    PT := T#1s);
   "Trigger_Run_FW_TF2" := "Delay_1s_4".Q AND NOT "Stop_Run_FW_TF2" AND NOT "TF2_Position_2";
   IF "Trigger_Run_FW_TF2" THEN "Being_TF2_FW" := TRUE; END_IF;
   "Delay_1s_5".TON(IN := (("AUTO_STATE" AND "TF2_Position_2" AND "SS Down XL Lift 5") OR "Trigger_Run_BW_TF2") AND ("RUN_TIME_PARAM".REQUEST_PICK_TYPE <> 1),
                    PT := T#1s);
   "Trigger_Run_BW_TF2" := "Delay_1s_5".Q AND NOT "Stop_Run_BW_TF2" AND NOT "TF2_Position_1";
   #_w1 := "Being_TF2_FW" AND "TF2_Position_2" AND "TF1_Position_2";
   "Delay_1s_6".TON(IN := #_w1, PT := T#1s);
   "Down_XL_Lift_5_Excute" := "Delay_1s_6".Q AND "SS Up XL Lift 5";
   IF "Down_XL_Lift_5_Excute" THEN
       "Mem_Status_2" := TRUE;
       "Being_TF2_FW" := FALSE;
   END_IF;
   "Lift_Rack_Down" := "Delay_1s_6".Q AND ("Axis_Lift".MasterData.Current_Position[0] = "ROBOT_PARAM".AxisLift_Position_1) AND ("Axis_Lift".MasterData.Current_Table_Point[1] = "ROBOT_PARAM".AxisLift_P1_Index);
   "Down_XL_Nâng Output" := "Delay_1s_6".Q;
   #_w2 := #_w1 AND NOT "Edge_140";   // rising edge
   "Edge_140" := #_w1;
   IF #_w2 THEN "SHIFT_RIGHT_DATA_AREA1_3"(); END_IF;
   IF "Mem_Status_2" AND "SS Down XL Lift 5" AND ("Axis_Lift".MasterData.Current_Position[0] = "ROBOT_PARAM".AxisLift_Position_2) AND ("Axis_Lift".MasterData.Current_Table_Point[1] = "ROBOT_PARAM".AxisLift_P2_Index) THEN
       "Begin_Tripping_1" := TRUE;
       "Mem_Status_2" := FALSE;
   END_IF;
   "Time_Tripping_Area3".TON(IN := "Begin_Tripping_1",
                           PT := "PROCESS_DATA_PARAMETER".Timer_Region1vs3,
                           ET => "PROCESS_DATA_PARAMETER".Current_TValue_Area_1);
   IF "Time_Tripping_Area3".Q AND NOT "Pause_Process" THEN "Begin_Tripping_1" := FALSE; END_IF;
   #_w3 := NOT "Begin_Tripping_1" AND "Edge_65";   // falling edge of "Begin_Tripping_1"
   "Edge_65" := "Begin_Tripping_1";
   "Edge_66" := (#_w3 OR "Edge_66") AND NOT "Stop_Delay_Temp_2";
   "Delay_1s_7".TON(IN := "Edge_66", PT := T#1s);
   "Stop_Delay_Temp_2" := "Delay_1s_7".Q;
   "Up_XL_Lift_5_Excute" := "Stop_Delay_Temp_2";
   "Lift_Rack_Up" := "Stop_Delay_Temp_2";
   "Up_XL_Nâng Output" := "Stop_Delay_Temp_2";
   IF "Stop_Delay_Temp_2" THEN "Tripping_Area3_Done" := TRUE; END_IF;
END_REGION

REGION Network 15: Trigger Run Lift 3 FW
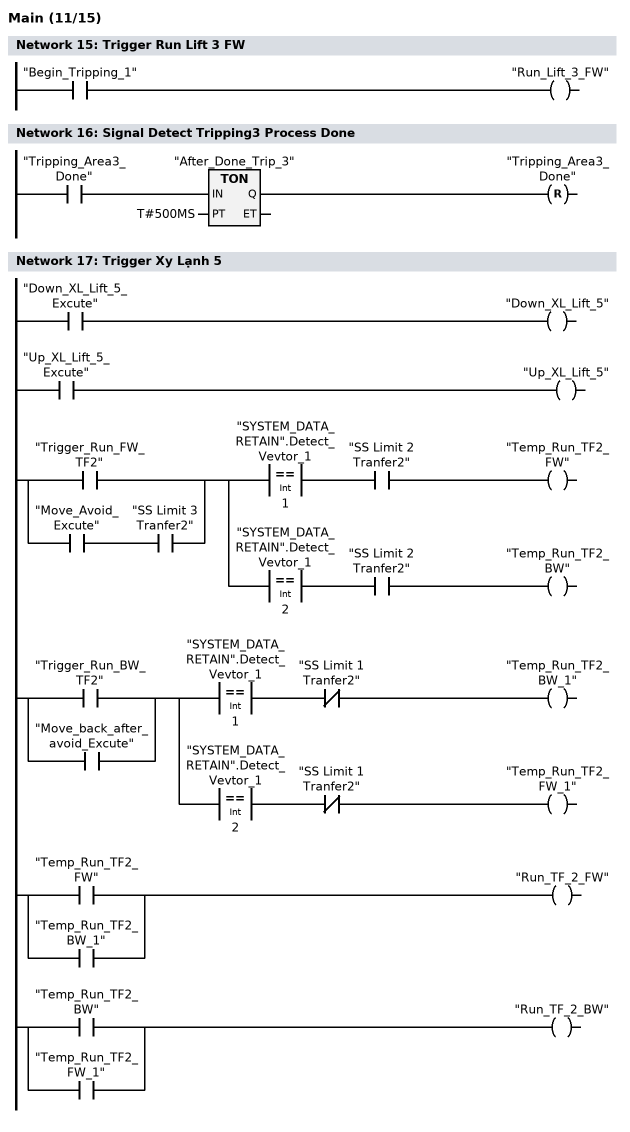
   RUNG wire#powerrail
      Contact( "Begin_Tripping_1" )
      Coil( "Run_Lift_3_FW" )
   END_RUNG
   // the same network as SCL:
   "Run_Lift_3_FW" := "Begin_Tripping_1";
END_REGION

REGION Network 16: Signal Detect Tripping3 Process Done
   "After_Done_Trip_3".TON(IN := "Tripping_Area3_Done", PT := T#500MS);
   IF "After_Done_Trip_3".Q THEN "Tripping_Area3_Done" := FALSE; END_IF;
END_REGION

REGION Network 17: Trigger Xy Lạnh 5
   RUNG wire#powerrail
      Contact( "Down_XL_Lift_5_Excute" )
      Coil( "Down_XL_Lift_5" )
   END_RUNG
   RUNG wire#powerrail
      Contact( "Up_XL_Lift_5_Excute" )
      Coil( "Up_XL_Lift_5" )
   END_RUNG
   RUNG wire#powerrail
      Contact( "Trigger_Run_FW_TF2" )
      wire#w1
      { S7_Templates := "SrcType := Int" } EQ_Contact(in1 := "SYSTEM_DATA_RETAIN".Detect_Vevtor_1, in2 := 1)
      Contact( "SS Limit 2 Tranfer2" )
      Coil( "Temp_Run_TF2_FW" )
   END_RUNG
   RUNG wire#powerrail
      Contact( "Move_Avoid_Excute" )
      Contact( "SS Limit 3 Tranfer2" )
   END_RUNG wire#w1
   RUNG wire#w1
      { S7_Templates := "SrcType := Int" } EQ_Contact(in1 := "SYSTEM_DATA_RETAIN".Detect_Vevtor_1, in2 := 2)
      Contact( "SS Limit 2 Tranfer2" )
      Coil( "Temp_Run_TF2_BW" )
   END_RUNG
   RUNG wire#powerrail
      Contact( "Trigger_Run_BW_TF2" )
      wire#w2
      { S7_Templates := "SrcType := Int" } EQ_Contact(in1 := "SYSTEM_DATA_RETAIN".Detect_Vevtor_1, in2 := 1)
      I_Contact( "SS Limit 1 Tranfer2" )
      Coil( "Temp_Run_TF2_BW_1" )
   END_RUNG
   RUNG wire#powerrail
      Contact( "Move_back_after_avoid_Excute" )
   END_RUNG wire#w2
   RUNG wire#w2
      { S7_Templates := "SrcType := Int" } EQ_Contact(in1 := "SYSTEM_DATA_RETAIN".Detect_Vevtor_1, in2 := 2)
      I_Contact( "SS Limit 1 Tranfer2" )
      Coil( "Temp_Run_TF2_FW_1" )
   END_RUNG
   RUNG wire#powerrail
      Contact( "Temp_Run_TF2_FW" )
      wire#w3
      Coil( "Run_TF_2_FW" )
   END_RUNG
   RUNG wire#powerrail
      Contact( "Temp_Run_TF2_BW_1" )
   END_RUNG wire#w3
   RUNG wire#powerrail
      Contact( "Temp_Run_TF2_BW" )
      wire#w4
      Coil( "Run_TF_2_BW" )
   END_RUNG
   RUNG wire#powerrail
      Contact( "Temp_Run_TF2_FW_1" )
   END_RUNG wire#w4
   // the same network as SCL:
   "Down_XL_Lift_5" := "Down_XL_Lift_5_Excute";
   "Up_XL_Lift_5" := "Up_XL_Lift_5_Excute";
   #_w1 := "Trigger_Run_FW_TF2" OR ("Move_Avoid_Excute" AND "SS Limit 3 Tranfer2");
   "Temp_Run_TF2_FW" := #_w1 AND ("SYSTEM_DATA_RETAIN".Detect_Vevtor_1 = 1) AND "SS Limit 2 Tranfer2";
   "Temp_Run_TF2_BW" := #_w1 AND ("SYSTEM_DATA_RETAIN".Detect_Vevtor_1 = 2) AND "SS Limit 2 Tranfer2";
   #_w2 := "Trigger_Run_BW_TF2" OR "Move_back_after_avoid_Excute";
   "Temp_Run_TF2_BW_1" := #_w2 AND ("SYSTEM_DATA_RETAIN".Detect_Vevtor_1 = 1) AND NOT "SS Limit 1 Tranfer2";
   "Temp_Run_TF2_FW_1" := #_w2 AND ("SYSTEM_DATA_RETAIN".Detect_Vevtor_1 = 2) AND NOT "SS Limit 1 Tranfer2";
   "Run_TF_2_FW" := "Temp_Run_TF2_FW" OR "Temp_Run_TF2_BW_1";
   "Run_TF_2_BW" := "Temp_Run_TF2_BW" OR "Temp_Run_TF2_FW_1";
END_REGION

REGION Network 18: Move TF2 to Avoid Robot
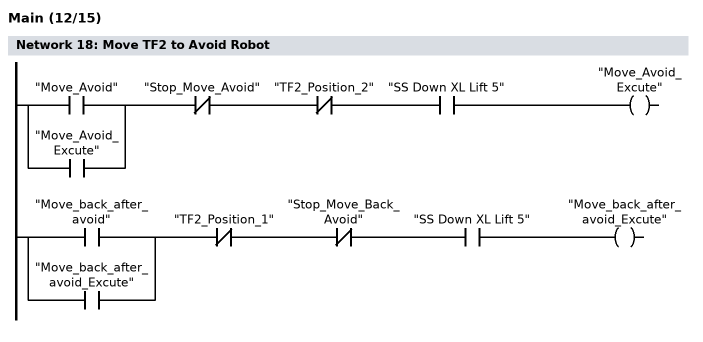
   RUNG wire#powerrail
      Contact( "Move_Avoid" )
      wire#w1
      I_Contact( "Stop_Move_Avoid" )
      I_Contact( "TF2_Position_2" )
      Contact( "SS Down XL Lift 5" )
      Coil( "Move_Avoid_Excute" )
   END_RUNG
   RUNG wire#powerrail
      Contact( "Move_Avoid_Excute" )
   END_RUNG wire#w1
   RUNG wire#powerrail
      Contact( "Move_back_after_avoid" )
      wire#w2
      I_Contact( "TF2_Position_1" )
      I_Contact( "Stop_Move_Back_Avoid" )
      Contact( "SS Down XL Lift 5" )
      Coil( "Move_back_after_avoid_Excute" )
   END_RUNG
   RUNG wire#powerrail
      Contact( "Move_back_after_avoid_Excute" )
   END_RUNG wire#w2
   // the same network as SCL:
   "Move_Avoid_Excute" := ("Move_Avoid" OR "Move_Avoid_Excute") AND NOT "Stop_Move_Avoid" AND NOT "TF2_Position_2" AND "SS Down XL Lift 5";
   "Move_back_after_avoid_Excute" := ("Move_back_after_avoid" OR "Move_back_after_avoid_Excute") AND NOT "TF2_Position_1" AND NOT "Stop_Move_Back_Avoid" AND "SS Down XL Lift 5";
END_REGION

REGION Network 19: Move Rack in Robot Area
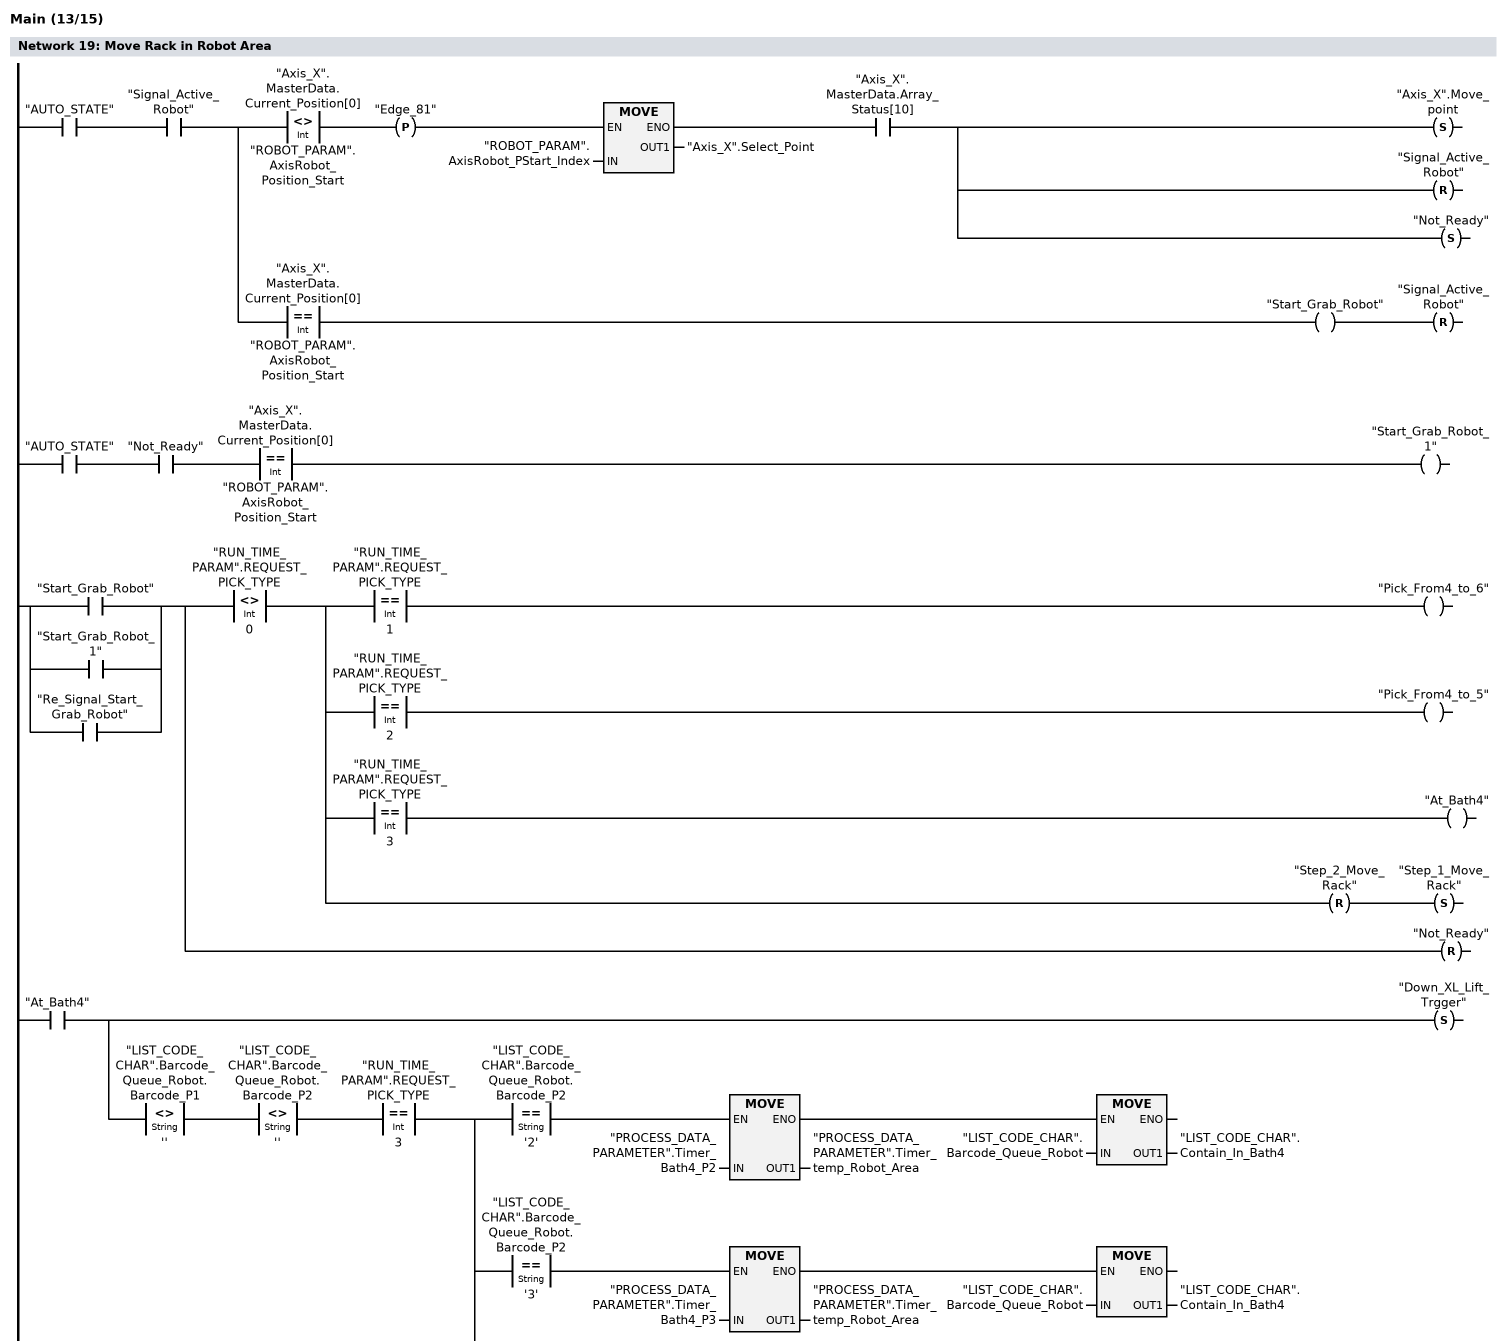
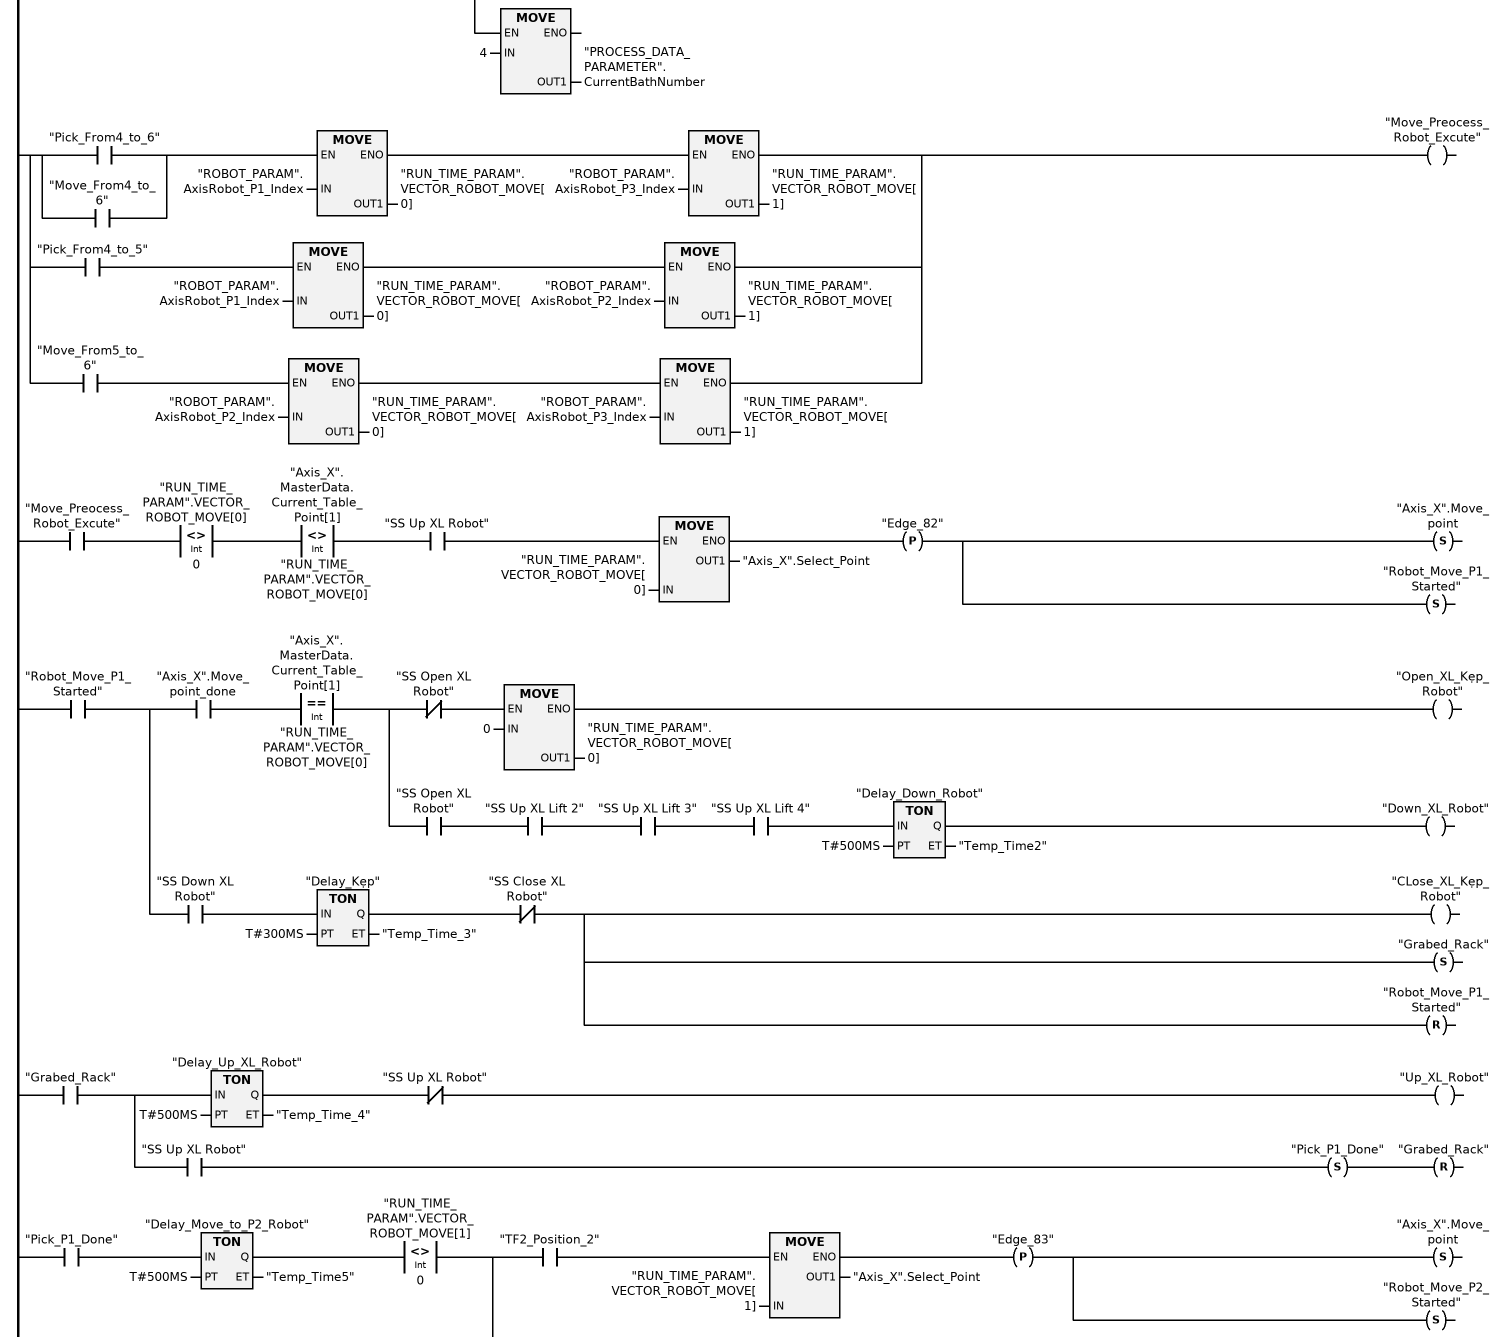
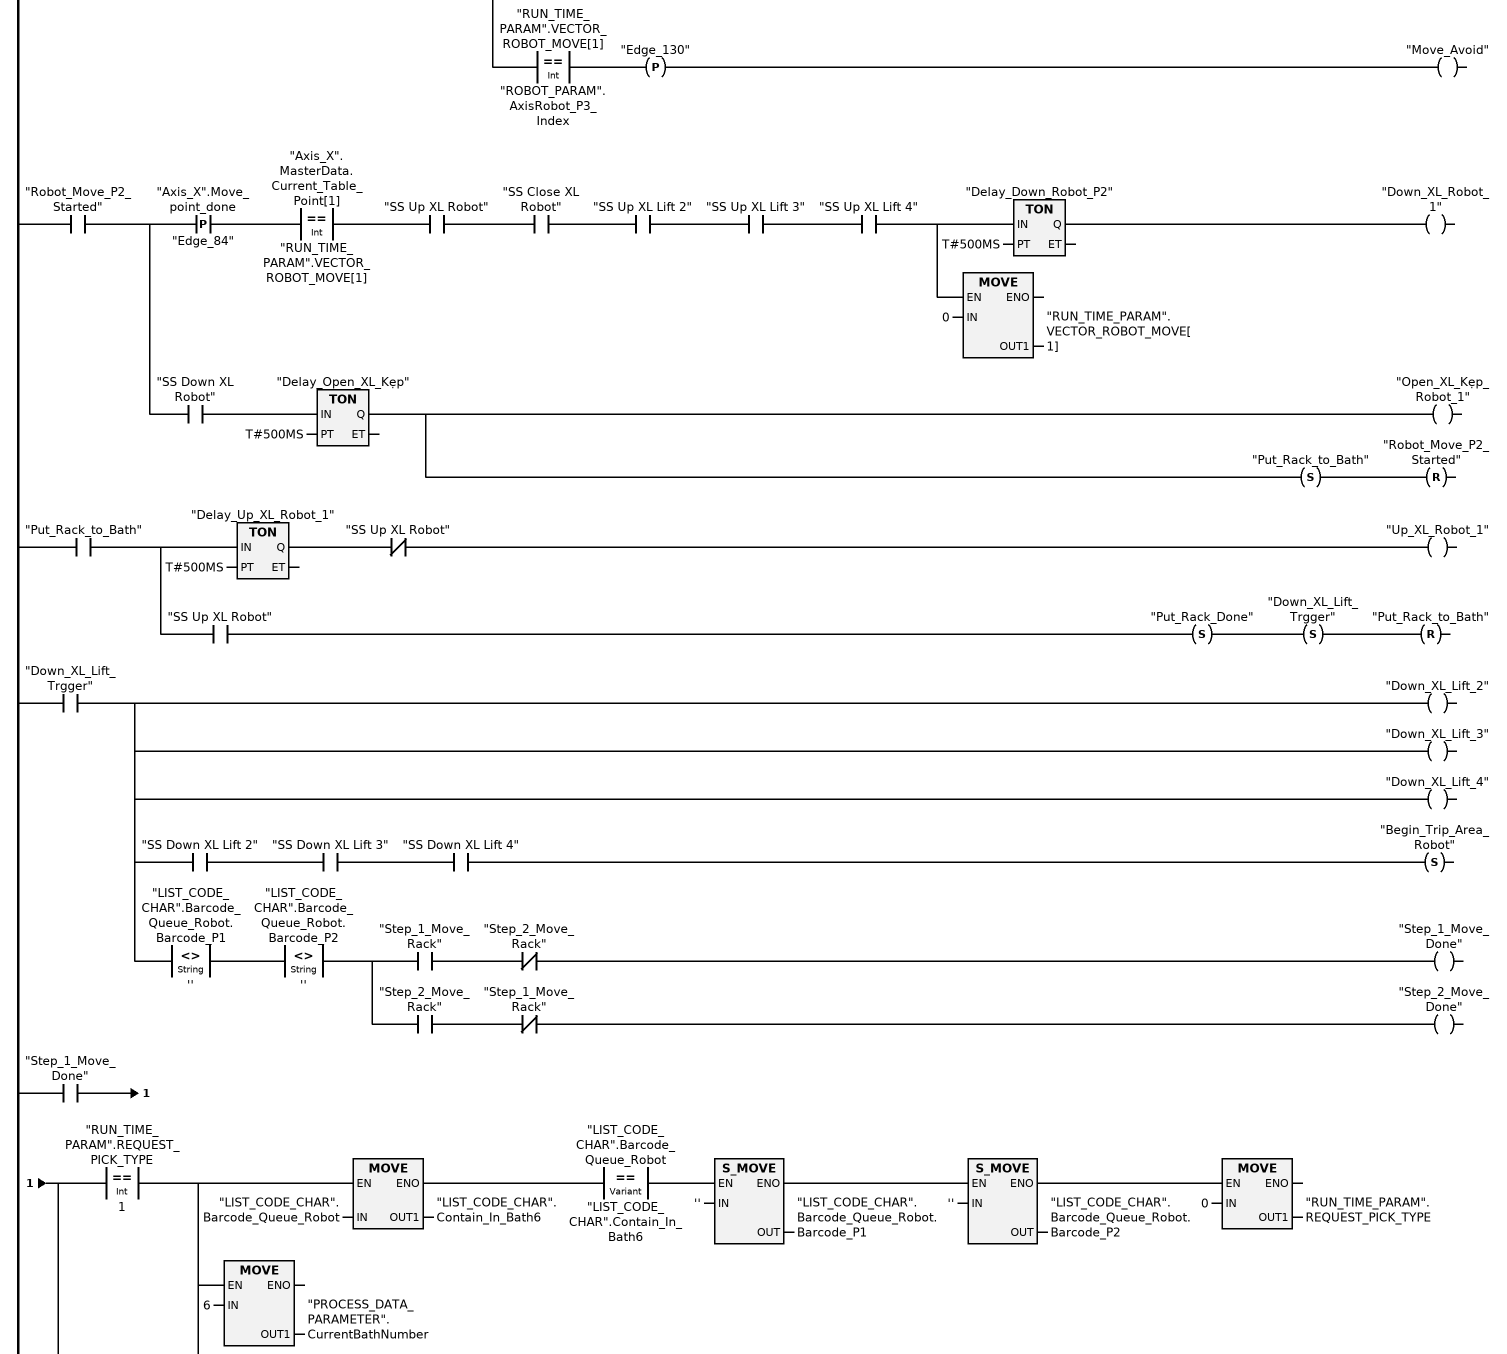
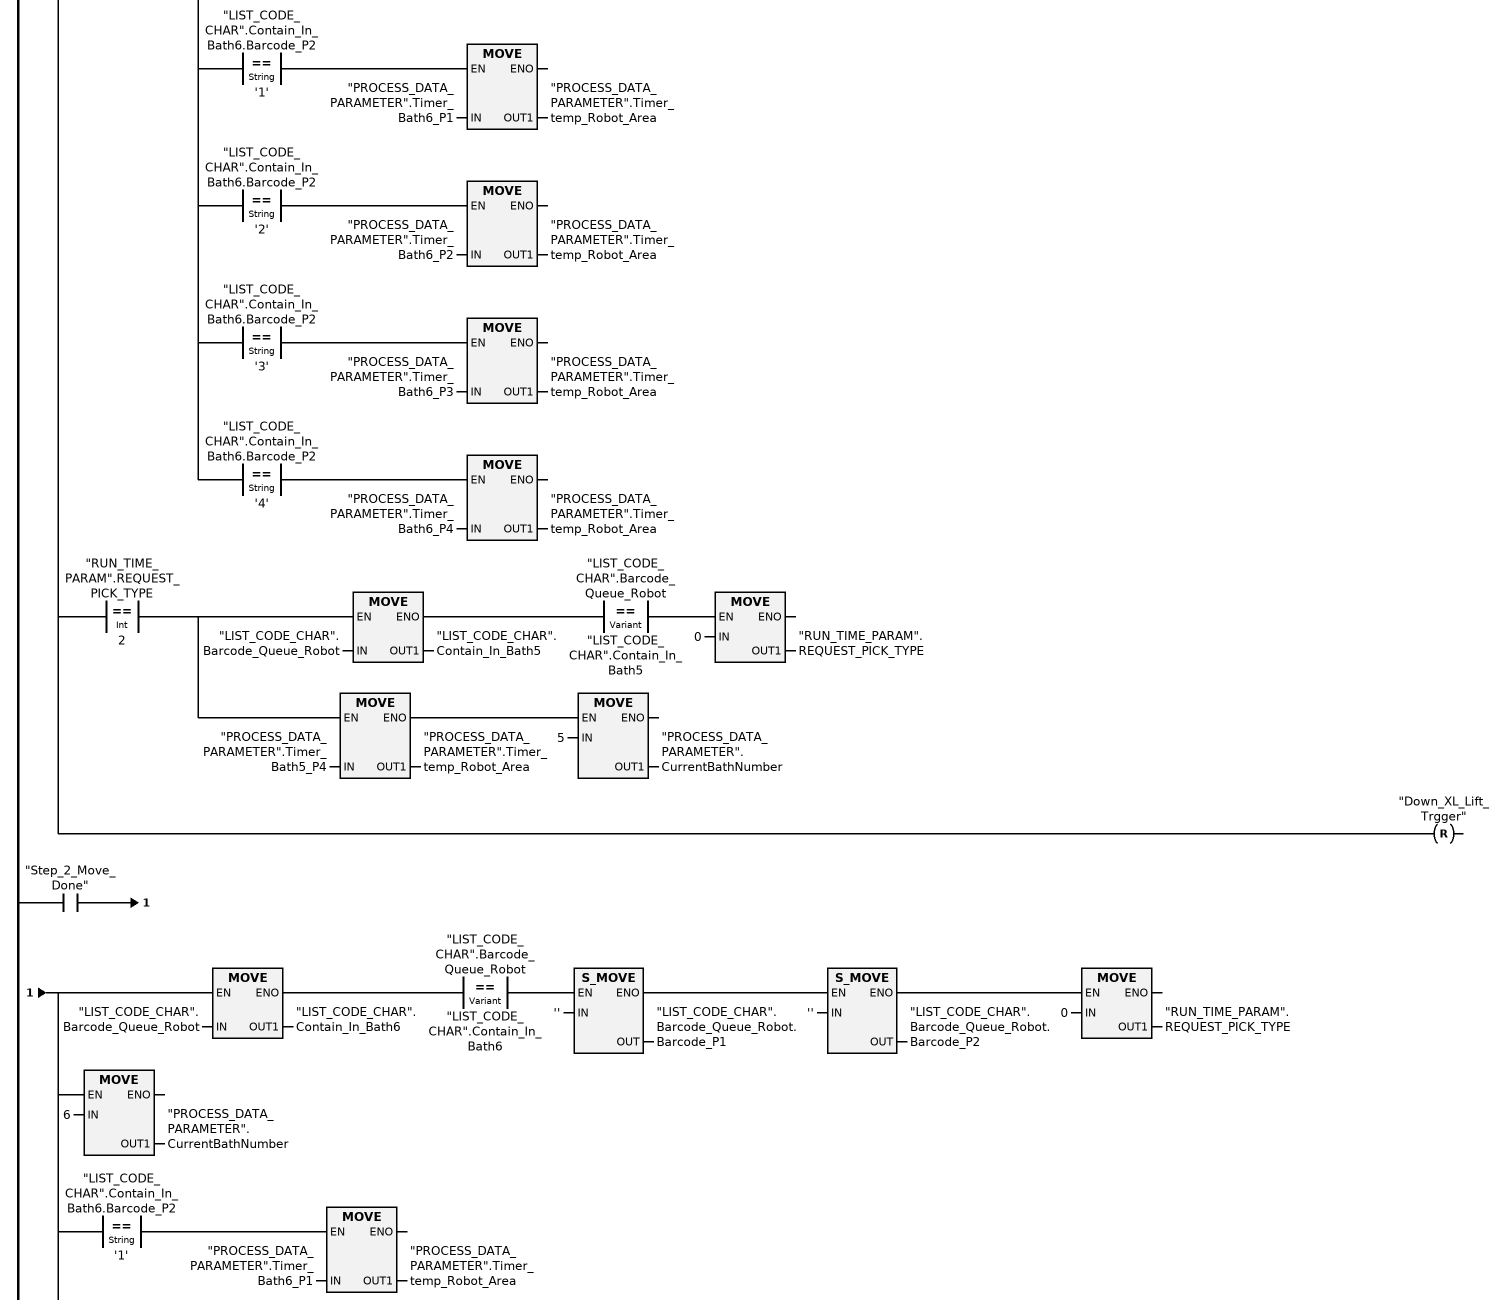
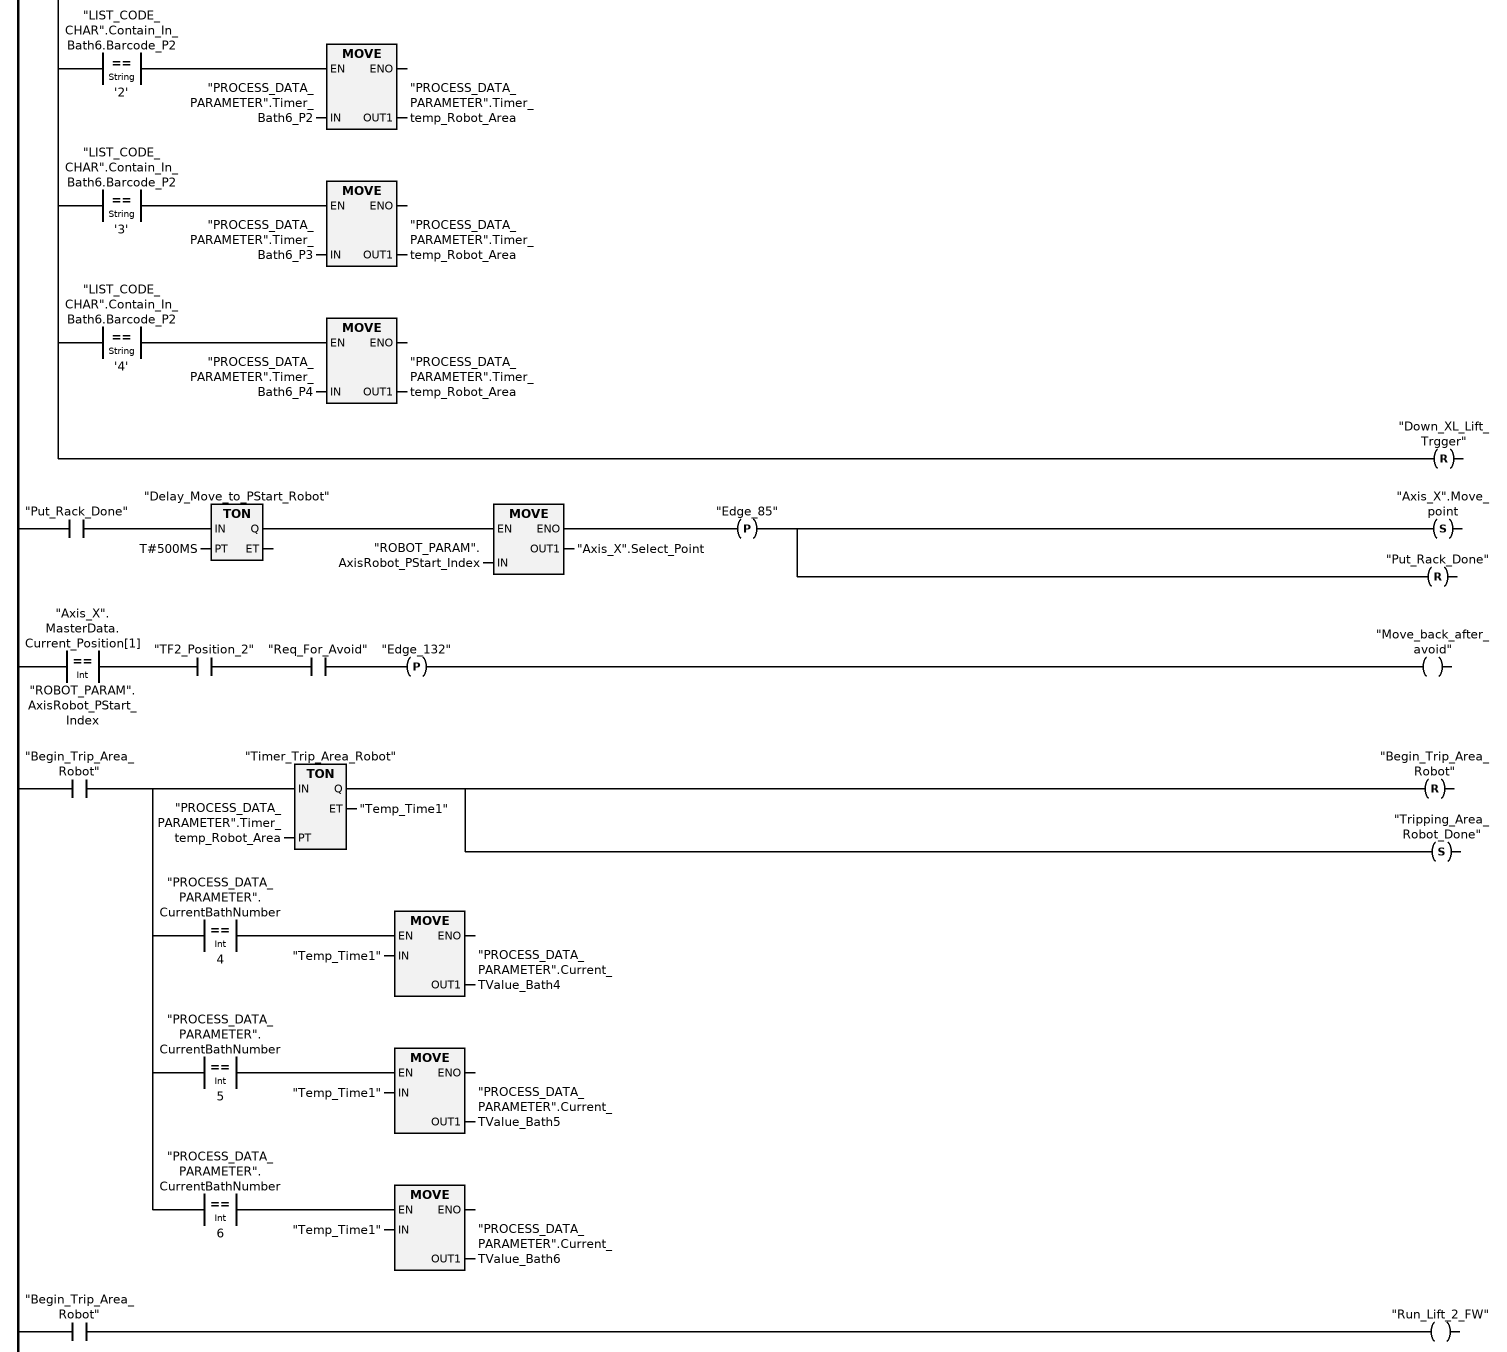
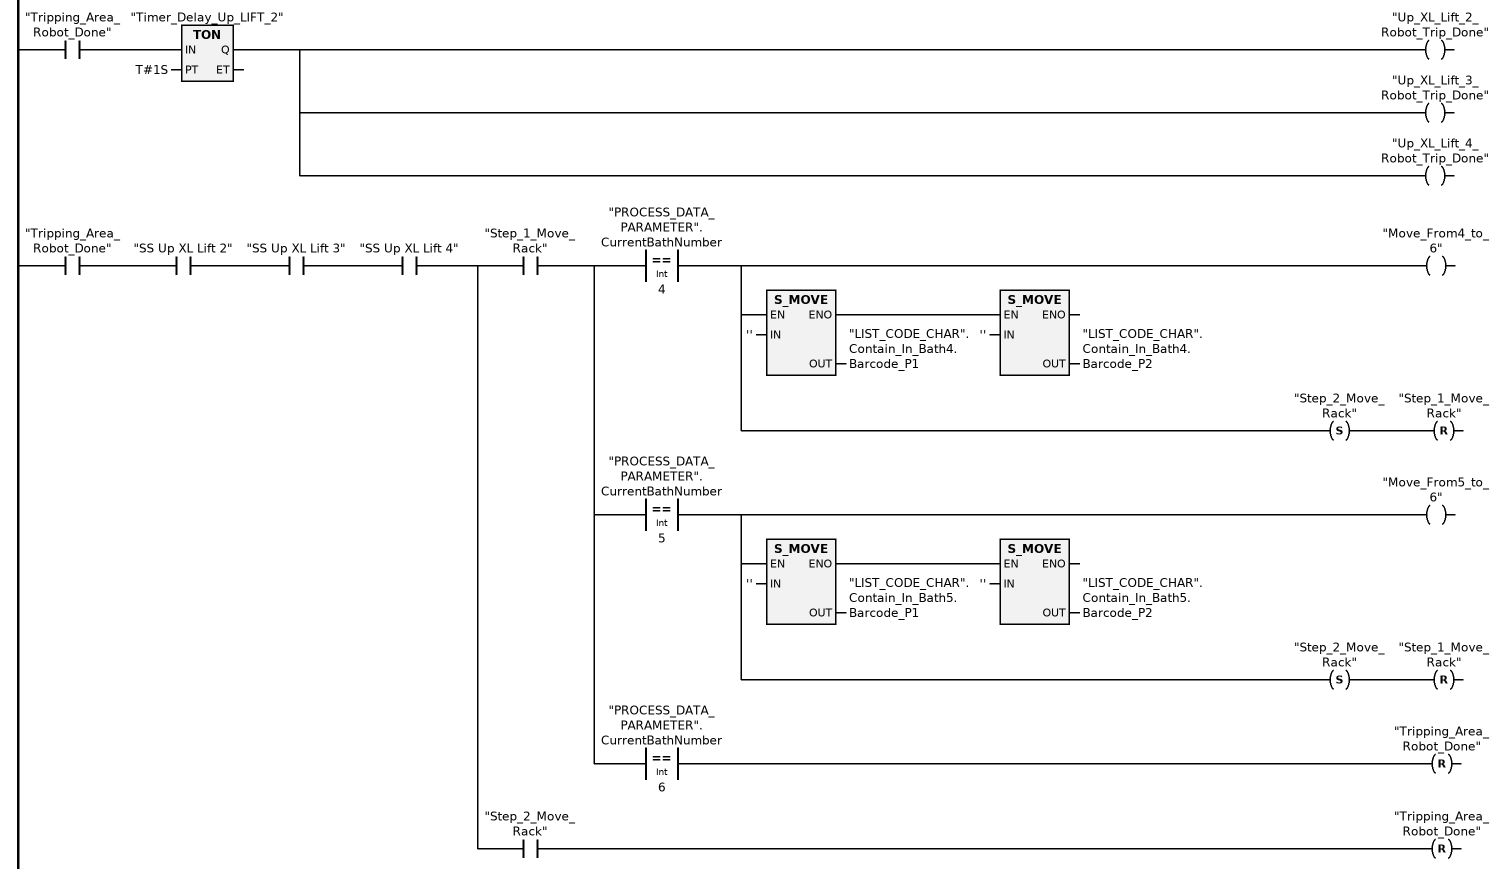
   // ENO of a box is taken as its EN; it also drops when the box reports an error
   #_w1 := "AUTO_STATE" AND "Signal_Active_Robot";
   #_w2 := #_w1 AND ("Axis_X".MasterData.Current_Position[0] <> "ROBOT_PARAM".AxisRobot_Position_Start);
   #_w3 := #_w2 AND NOT "Edge_81";   // rising edge
   "Edge_81" := #_w2;
   IF #_w3 THEN "Axis_X".Select_Point := "ROBOT_PARAM".AxisRobot_PStart_Index; END_IF;
   IF #_w3 AND "Axis_X".MasterData.Array_Status[10] THEN
       "Axis_X".Move_point := TRUE;
       "Signal_Active_Robot" := FALSE;
       "Not_Ready" := TRUE;
   END_IF;
   "Start_Grab_Robot" := #_w1 AND ("Axis_X".MasterData.Current_Position[0] = "ROBOT_PARAM".AxisRobot_Position_Start);
   IF "Start_Grab_Robot" THEN "Signal_Active_Robot" := FALSE; END_IF;
   "Start_Grab_Robot_1" := "AUTO_STATE" AND "Not_Ready" AND ("Axis_X".MasterData.Current_Position[0] = "ROBOT_PARAM".AxisRobot_Position_Start);
   #_w4 := "Start_Grab_Robot" OR "Start_Grab_Robot_1" OR "Re_Signal_Start_Grab_Robot";
   #_w5 := #_w4 AND ("RUN_TIME_PARAM".REQUEST_PICK_TYPE <> 0);
   "Pick_From4_to_6" := #_w5 AND ("RUN_TIME_PARAM".REQUEST_PICK_TYPE = 1);
   "Pick_From4_to_5" := #_w5 AND ("RUN_TIME_PARAM".REQUEST_PICK_TYPE = 2);
   "At_Bath4" := #_w5 AND ("RUN_TIME_PARAM".REQUEST_PICK_TYPE = 3);
   IF #_w5 THEN
       "Step_2_Move_Rack" := FALSE;
       "Step_1_Move_Rack" := TRUE;
   END_IF;
   IF #_w4 THEN "Not_Ready" := FALSE; END_IF;
   IF "At_Bath4" THEN "Down_XL_Lift_Trgger" := TRUE; END_IF;
   #_w6 := "At_Bath4" AND ("LIST_CODE_CHAR".Barcode_Queue_Robot.Barcode_P1 <> '') AND ("LIST_CODE_CHAR".Barcode_Queue_Robot.Barcode_P2 <> '') AND ("RUN_TIME_PARAM".REQUEST_PICK_TYPE = 3);
   IF #_w6 AND ("LIST_CODE_CHAR".Barcode_Queue_Robot.Barcode_P2 = '2') THEN
       "PROCESS_DATA_PARAMETER".Timer_temp_Robot_Area := "PROCESS_DATA_PARAMETER".Timer_Bath4_P2;
       "LIST_CODE_CHAR".Contain_In_Bath4 := "LIST_CODE_CHAR".Barcode_Queue_Robot;
   END_IF;
   IF #_w6 AND ("LIST_CODE_CHAR".Barcode_Queue_Robot.Barcode_P2 = '3') THEN
       "PROCESS_DATA_PARAMETER".Timer_temp_Robot_Area := "PROCESS_DATA_PARAMETER".Timer_Bath4_P3;
       "LIST_CODE_CHAR".Contain_In_Bath4 := "LIST_CODE_CHAR".Barcode_Queue_Robot;
   END_IF;
   IF #_w6 THEN "PROCESS_DATA_PARAMETER".CurrentBathNumber := 4; END_IF;
   #_w7 := "Pick_From4_to_6" OR "Move_From4_to_6";
   IF #_w7 THEN
       "RUN_TIME_PARAM".VECTOR_ROBOT_MOVE[0] := "ROBOT_PARAM".AxisRobot_P1_Index;
       "RUN_TIME_PARAM".VECTOR_ROBOT_MOVE[1] := "ROBOT_PARAM".AxisRobot_P3_Index;
   END_IF;
   IF "Pick_From4_to_5" THEN
       "RUN_TIME_PARAM".VECTOR_ROBOT_MOVE[0] := "ROBOT_PARAM".AxisRobot_P1_Index;
       "RUN_TIME_PARAM".VECTOR_ROBOT_MOVE[1] := "ROBOT_PARAM".AxisRobot_P2_Index;
   END_IF;
   IF "Move_From5_to_6" THEN
       "RUN_TIME_PARAM".VECTOR_ROBOT_MOVE[0] := "ROBOT_PARAM".AxisRobot_P2_Index;
       "RUN_TIME_PARAM".VECTOR_ROBOT_MOVE[1] := "ROBOT_PARAM".AxisRobot_P3_Index;
   END_IF;
   "Move_Preocess_Robot_Excute" := #_w7 OR "Pick_From4_to_5" OR "Move_From5_to_6";
   #_w8 := "Move_Preocess_Robot_Excute" AND ("RUN_TIME_PARAM".VECTOR_ROBOT_MOVE[0] <> 0) AND ("Axis_X".MasterData.Current_Table_Point[1] <> "RUN_TIME_PARAM".VECTOR_ROBOT_MOVE[0]) AND "SS Up XL Robot";
   IF #_w8 THEN "Axis_X".Select_Point := "RUN_TIME_PARAM".VECTOR_ROBOT_MOVE[0]; END_IF;
   #_w9 := #_w8 AND NOT "Edge_82";   // rising edge
   "Edge_82" := #_w8;
   IF #_w9 THEN
       "Axis_X".Move_point := TRUE;
       "Robot_Move_P1_Started" := TRUE;
   END_IF;
   #_w10 := "Robot_Move_P1_Started" AND "Axis_X".Move_point_done AND ("Axis_X".MasterData.Current_Table_Point[1] = "RUN_TIME_PARAM".VECTOR_ROBOT_MOVE[0]);
   #_w11 := #_w10 AND NOT "SS Open XL Robot";
   IF #_w11 THEN "RUN_TIME_PARAM".VECTOR_ROBOT_MOVE[0] := 0; END_IF;
   "Open_XL_Kẹp_Robot" := #_w11;
   "Delay_Down_Robot".TON(IN := #_w10 AND "SS Open XL Robot" AND "SS Up XL Lift 2" AND "SS Up XL Lift 3" AND "SS Up XL Lift 4",
                          PT := T#500MS,
                          ET => "Temp_Time2");
   "Down_XL_Robot" := "Delay_Down_Robot".Q;
   "Delay_Kẹp".TON(IN := "Robot_Move_P1_Started" AND "SS Down XL Robot", PT := T#300MS, ET => "Temp_Time_3");
   "CLose_XL_Kẹp_Robot" := "Delay_Kẹp".Q AND NOT "SS Close XL Robot";
   IF "CLose_XL_Kẹp_Robot" THEN
       "Grabed_Rack" := TRUE;
       "Robot_Move_P1_Started" := FALSE;
   END_IF;
   "Delay_Up_XL_Robot".TON(IN := "Grabed_Rack", PT := T#500MS, ET => "Temp_Time_4");
   "Up_XL_Robot" := "Delay_Up_XL_Robot".Q AND NOT "SS Up XL Robot";
   IF "Grabed_Rack" AND "SS Up XL Robot" THEN
       "Pick_P1_Done" := TRUE;
       "Grabed_Rack" := FALSE;
   END_IF;
   "Delay_Move_to_P2_Robot".TON(IN := "Pick_P1_Done", PT := T#500MS, ET => "Temp_Time5");
   #_w12 := "Delay_Move_to_P2_Robot".Q AND ("RUN_TIME_PARAM".VECTOR_ROBOT_MOVE[1] <> 0);
   #_w13 := #_w12 AND "TF2_Position_2";
   IF #_w13 THEN "Axis_X".Select_Point := "RUN_TIME_PARAM".VECTOR_ROBOT_MOVE[1]; END_IF;
   #_w14 := #_w13 AND NOT "Edge_83";   // rising edge
   "Edge_83" := #_w13;
   IF #_w14 THEN
       "Axis_X".Move_point := TRUE;
       "Robot_Move_P2_Started" := TRUE;
   END_IF;
   #_w15 := #_w12 AND ("RUN_TIME_PARAM".VECTOR_ROBOT_MOVE[1] = "ROBOT_PARAM".AxisRobot_P3_Index);
   #_w16 := #_w15 AND NOT "Edge_130";   // rising edge
   "Edge_130" := #_w15;
   "Move_Avoid" := #_w16;
   #_w17 := "Robot_Move_P2_Started" AND "Axis_X".Move_point_done AND NOT "Edge_84";   // rising edge of "Axis_X".Move_point_done
   "Edge_84" := "Axis_X".Move_point_done;
   #_w18 := #_w17 AND ("Axis_X".MasterData.Current_Table_Point[1] = "RUN_TIME_PARAM".VECTOR_ROBOT_MOVE[1]) AND "SS Up XL Robot" AND "SS Close XL Robot" AND "SS Up XL Lift 2" AND "SS Up XL Lift 3" AND "SS Up XL Lift 4";
   "Delay_Down_Robot_P2".TON(IN := #_w18, PT := T#500MS);
   "Down_XL_Robot_1" := "Delay_Down_Robot_P2".Q;
   IF #_w18 THEN "RUN_TIME_PARAM".VECTOR_ROBOT_MOVE[1] := 0; END_IF;
   "Delay_Open_XL_Kẹp".TON(IN := "Robot_Move_P2_Started" AND "SS Down XL Robot", PT := T#500MS);
   "Open_XL_Kẹp_Robot_1" := "Delay_Open_XL_Kẹp".Q;
   IF "Delay_Open_XL_Kẹp".Q THEN
       "Put_Rack_to_Bath" := TRUE;
       "Robot_Move_P2_Started" := FALSE;
   END_IF;
   "Delay_Up_XL_Robot_1".TON(IN := "Put_Rack_to_Bath", PT := T#500MS);
   "Up_XL_Robot_1" := "Delay_Up_XL_Robot_1".Q AND NOT "SS Up XL Robot";
   IF "Put_Rack_to_Bath" AND "SS Up XL Robot" THEN
       "Put_Rack_Done" := TRUE;
       "Down_XL_Lift_Trgger" := TRUE;
       "Put_Rack_to_Bath" := FALSE;
   END_IF;
   "Down_XL_Lift_2" := "Down_XL_Lift_Trgger";
   "Down_XL_Lift_3" := "Down_XL_Lift_Trgger";
   "Down_XL_Lift_4" := "Down_XL_Lift_Trgger";
   IF "Down_XL_Lift_Trgger" AND "SS Down XL Lift 2" AND "SS Down XL Lift 3" AND "SS Down XL Lift 4" THEN
       "Begin_Trip_Area_Robot" := TRUE;
   END_IF;
   #_w19 := "Down_XL_Lift_Trgger" AND ("LIST_CODE_CHAR".Barcode_Queue_Robot.Barcode_P1 <> '') AND ("LIST_CODE_CHAR".Barcode_Queue_Robot.Barcode_P2 <> '');
   "Step_1_Move_Done" := #_w19 AND "Step_1_Move_Rack" AND NOT "Step_2_Move_Rack";
   "Step_2_Move_Done" := #_w19 AND "Step_2_Move_Rack" AND NOT "Step_1_Move_Rack";
   #_w20 := "Step_1_Move_Done" AND ("RUN_TIME_PARAM".REQUEST_PICK_TYPE = 1);
   IF #_w20 THEN "LIST_CODE_CHAR".Contain_In_Bath6 := "LIST_CODE_CHAR".Barcode_Queue_Robot; END_IF;
   #_w21 := #_w20 AND ("LIST_CODE_CHAR".Barcode_Queue_Robot = "LIST_CODE_CHAR".Contain_In_Bath6);
   IF #_w21 THEN
       "LIST_CODE_CHAR".Barcode_Queue_Robot.Barcode_P1 := '';
       "LIST_CODE_CHAR".Barcode_Queue_Robot.Barcode_P2 := '';
       "RUN_TIME_PARAM".REQUEST_PICK_TYPE := 0;
   END_IF;
   IF #_w20 THEN "PROCESS_DATA_PARAMETER".CurrentBathNumber := 6; END_IF;
   IF #_w20 AND ("LIST_CODE_CHAR".Contain_In_Bath6.Barcode_P2 = '1') THEN
       "PROCESS_DATA_PARAMETER".Timer_temp_Robot_Area := "PROCESS_DATA_PARAMETER".Timer_Bath6_P1;
   END_IF;
   IF #_w20 AND ("LIST_CODE_CHAR".Contain_In_Bath6.Barcode_P2 = '2') THEN
       "PROCESS_DATA_PARAMETER".Timer_temp_Robot_Area := "PROCESS_DATA_PARAMETER".Timer_Bath6_P2;
   END_IF;
   IF #_w20 AND ("LIST_CODE_CHAR".Contain_In_Bath6.Barcode_P2 = '3') THEN
       "PROCESS_DATA_PARAMETER".Timer_temp_Robot_Area := "PROCESS_DATA_PARAMETER".Timer_Bath6_P3;
   END_IF;
   IF #_w20 AND ("LIST_CODE_CHAR".Contain_In_Bath6.Barcode_P2 = '4') THEN
       "PROCESS_DATA_PARAMETER".Timer_temp_Robot_Area := "PROCESS_DATA_PARAMETER".Timer_Bath6_P4;
   END_IF;
   #_w22 := "Step_1_Move_Done" AND ("RUN_TIME_PARAM".REQUEST_PICK_TYPE = 2);
   IF #_w22 THEN "LIST_CODE_CHAR".Contain_In_Bath5 := "LIST_CODE_CHAR".Barcode_Queue_Robot; END_IF;
   IF #_w22 AND ("LIST_CODE_CHAR".Barcode_Queue_Robot = "LIST_CODE_CHAR".Contain_In_Bath5) THEN
       "RUN_TIME_PARAM".REQUEST_PICK_TYPE := 0;
   END_IF;
   IF #_w22 THEN
       "PROCESS_DATA_PARAMETER".Timer_temp_Robot_Area := "PROCESS_DATA_PARAMETER".Timer_Bath5_P4;
       "PROCESS_DATA_PARAMETER".CurrentBathNumber := 5;
   END_IF;
   IF "Step_1_Move_Done" THEN "Down_XL_Lift_Trgger" := FALSE; END_IF;
   IF "Step_2_Move_Done" THEN
       "LIST_CODE_CHAR".Contain_In_Bath6 := "LIST_CODE_CHAR".Barcode_Queue_Robot;
   END_IF;
   #_w23 := "Step_2_Move_Done" AND ("LIST_CODE_CHAR".Barcode_Queue_Robot = "LIST_CODE_CHAR".Contain_In_Bath6);
   IF #_w23 THEN
       "LIST_CODE_CHAR".Barcode_Queue_Robot.Barcode_P1 := '';
       "LIST_CODE_CHAR".Barcode_Queue_Robot.Barcode_P2 := '';
       "RUN_TIME_PARAM".REQUEST_PICK_TYPE := 0;
   END_IF;
   IF "Step_2_Move_Done" THEN "PROCESS_DATA_PARAMETER".CurrentBathNumber := 6; END_IF;
   IF "Step_2_Move_Done" AND ("LIST_CODE_CHAR".Contain_In_Bath6.Barcode_P2 = '1') THEN
       "PROCESS_DATA_PARAMETER".Timer_temp_Robot_Area := "PROCESS_DATA_PARAMETER".Timer_Bath6_P1;
   END_IF;
   IF "Step_2_Move_Done" AND ("LIST_CODE_CHAR".Contain_In_Bath6.Barcode_P2 = '2') THEN
       "PROCESS_DATA_PARAMETER".Timer_temp_Robot_Area := "PROCESS_DATA_PARAMETER".Timer_Bath6_P2;
   END_IF;
   IF "Step_2_Move_Done" AND ("LIST_CODE_CHAR".Contain_In_Bath6.Barcode_P2 = '3') THEN
       "PROCESS_DATA_PARAMETER".Timer_temp_Robot_Area := "PROCESS_DATA_PARAMETER".Timer_Bath6_P3;
   END_IF;
   IF "Step_2_Move_Done" AND ("LIST_CODE_CHAR".Contain_In_Bath6.Barcode_P2 = '4') THEN
       "PROCESS_DATA_PARAMETER".Timer_temp_Robot_Area := "PROCESS_DATA_PARAMETER".Timer_Bath6_P4;
   END_IF;
   IF "Step_2_Move_Done" THEN "Down_XL_Lift_Trgger" := FALSE; END_IF;
   "Delay_Move_to_PStart_Robot".TON(IN := "Put_Rack_Done", PT := T#500MS);
   IF "Delay_Move_to_PStart_Robot".Q THEN
       "Axis_X".Select_Point := "ROBOT_PARAM".AxisRobot_PStart_Index;
   END_IF;
   #_w24 := "Delay_Move_to_PStart_Robot".Q AND NOT "Edge_85";   // rising edge
   "Edge_85" := "Delay_Move_to_PStart_Robot".Q;
   IF #_w24 THEN
       "Axis_X".Move_point := TRUE;
       "Put_Rack_Done" := FALSE;
   END_IF;
   #_w25 := ("Axis_X".MasterData.Current_Position[1] = "ROBOT_PARAM".AxisRobot_PStart_Index) AND "TF2_Position_2" AND "Req_For_Avoid";
   #_w26 := #_w25 AND NOT "Edge_132";   // rising edge
   "Edge_132" := #_w25;
   "Move_back_after_avoid" := #_w26;
   "Timer_Trip_Area_Robot".TON(IN := "Begin_Trip_Area_Robot",
                           PT := "PROCESS_DATA_PARAMETER".Timer_temp_Robot_Area,
                           ET => "Temp_Time1");
   #_w27 := "Begin_Trip_Area_Robot";
   IF "Timer_Trip_Area_Robot".Q THEN
       "Begin_Trip_Area_Robot" := FALSE;
       "Tripping_Area_Robot_Done" := TRUE;
   END_IF;
   IF #_w27 AND ("PROCESS_DATA_PARAMETER".CurrentBathNumber = 4) THEN
       "PROCESS_DATA_PARAMETER".Current_TValue_Bath4 := "Temp_Time1";
   END_IF;
   IF #_w27 AND ("PROCESS_DATA_PARAMETER".CurrentBathNumber = 5) THEN
       "PROCESS_DATA_PARAMETER".Current_TValue_Bath5 := "Temp_Time1";
   END_IF;
   IF #_w27 AND ("PROCESS_DATA_PARAMETER".CurrentBathNumber = 6) THEN
       "PROCESS_DATA_PARAMETER".Current_TValue_Bath6 := "Temp_Time1";
   END_IF;
   "Run_Lift_2_FW" := "Begin_Trip_Area_Robot";
   "Timer_Delay_Up_LIFT_2".TON(IN := "Tripping_Area_Robot_Done", PT := T#1S);
   "Up_XL_Lift_2_Robot_Trip_Done" := "Timer_Delay_Up_LIFT_2".Q;
   "Up_XL_Lift_3_Robot_Trip_Done" := "Timer_Delay_Up_LIFT_2".Q;
   "Up_XL_Lift_4_Robot_Trip_Done" := "Timer_Delay_Up_LIFT_2".Q;
   #_w28 := "Tripping_Area_Robot_Done" AND "SS Up XL Lift 2" AND "SS Up XL Lift 3" AND "SS Up XL Lift 4";
   #_w29 := #_w28 AND "Step_1_Move_Rack";
   "Move_From4_to_6" := #_w29 AND ("PROCESS_DATA_PARAMETER".CurrentBathNumber = 4);
   IF "Move_From4_to_6" THEN
       "LIST_CODE_CHAR".Contain_In_Bath4.Barcode_P1 := '';
       "LIST_CODE_CHAR".Contain_In_Bath4.Barcode_P2 := '';
       "Step_2_Move_Rack" := TRUE;
       "Step_1_Move_Rack" := FALSE;
   END_IF;
   "Move_From5_to_6" := #_w29 AND ("PROCESS_DATA_PARAMETER".CurrentBathNumber = 5);
   IF "Move_From5_to_6" THEN
       "LIST_CODE_CHAR".Contain_In_Bath5.Barcode_P1 := '';
       "LIST_CODE_CHAR".Contain_In_Bath5.Barcode_P2 := '';
       "Step_2_Move_Rack" := TRUE;
       "Step_1_Move_Rack" := FALSE;
   END_IF;
   IF #_w29 AND ("PROCESS_DATA_PARAMETER".CurrentBathNumber = 6) THEN
       "Tripping_Area_Robot_Done" := FALSE;
   END_IF;
   IF #_w28 AND "Step_2_Move_Rack" THEN "Tripping_Area_Robot_Done" := FALSE; END_IF;
END_REGION

REGION Network 20: Servo Lift Rack
